// NeuroPLC — Auto-generated IEC 61131-3 SCL
// Graph: mlp | Target: S71200Backend
// Work memory: 75KB | LUT points: 15
// Nodes: 8 | Ops: {'matmul': 4, 'standard_act': 2, 'softmax': 1, 'argmax': 1}


DATA_BLOCK "NeuroPLC_Weights"
{ S7_Optimized_Access := 'TRUE' }
VERSION : 0.1
NON_RETAIN

   // MatMul 'fc0': W(32×28) + b(32)
   w0 : Array[0..927] of Real :=
    -0.1798824, -0.3872150, 0.2042089, 0.0008930, 0.2428655, -0.4397896, 0.1184483, 0.1381282,
    0.0788599, -0.0335890, 0.3613543, -0.3164068, -0.3411417, -0.1364205, -0.3815753, 0.0980671,
    0.0654392, -0.0128052, 0.1792001, -0.1123531, -0.3475231, 0.1503572, -0.0112453, 0.1635510,
    0.1945115, 0.0545633, 0.4145930, -0.3514731, 0.0562777, 0.1928302, -0.1798587, -0.2800348,
    0.1141335, 0.3939485, -0.1134134, -0.3142068, 0.0689715, 0.2764131, -0.3031770, 0.3679943,
    0.0101338, -0.2268585, -0.1187166, 0.4428278, 0.1090220, -0.1324965, -0.4557532, 0.0609620,
    0.2945257, -0.4372934, -0.2674722, 0.2719050, -0.1746262, -0.4510055, -0.2193495, -0.0693161,
    -0.4133973, 0.4597808, 0.3899092, 0.2787638, 0.2211191, -0.2335375, -0.1846817, -0.1514431,
    0.2064924, -0.2602171, 0.2605978, 0.0973142, -0.3398410, -0.4581998, -0.2922807, -0.4378471,
    0.1851701, 0.3957313, 0.2401366, -0.3643467, -0.3337855, 0.0937589, -0.4046761, 0.3407934,
    -0.0060355, 0.0787147, -0.1516189, 0.4190823, 0.1787451, 0.3653978, -0.2563615, -0.3936344,
    -0.4418108, 0.0399490, -0.0161863, 0.3734512, -0.1328384, -0.3586327, 0.0832884, 0.3898760,
    0.0422331, 0.3219765, 0.4136791, 0.4541050, -0.2442907, 0.1221973, -0.3816552, -0.4393946,
    0.4381784, -0.3776088, -0.0355673, 0.0102973, 0.2750401, 0.4402033, -0.0992043, 0.3619939,
    -0.3341672, 0.3641900, 0.0646533, -0.0329038, -0.0519513, 0.4624202, 0.3974202, -0.4135628,
    -0.1883360, 0.1582608, -0.3120753, 0.3418854, -0.1363405, 0.3182234, 0.3987226, -0.2059435,
    0.1484261, 0.1623119, -0.1709910, 0.4116440, 0.4557955, 0.0284270, -0.0647671, 0.4628531,
    -0.4262170, -0.0586162, -0.0261355, 0.3885587, -0.0612076, 0.3511490, -0.4214011, 0.2382351,
    -0.0945188, 0.3279837, -0.4308659, 0.2451999, -0.3082491, -0.0678181, -0.2555402, 0.4352351,
    0.3423308, 0.1892392, -0.4397568, 0.0099074, 0.2687223, -0.4212352, -0.0019993, 0.0687157,
    0.0788325, 0.4018357, 0.4349293, -0.3687074, 0.2395242, 0.3815289, -0.4383415, -0.0245892,
    0.2103941, 0.0996155, 0.1315596, 0.1972513, 0.0423024, 0.3604410, 0.2333128, 0.2266048,
    0.0023598, 0.4544540, -0.2608073, -0.0723180, 0.3625811, 0.1550818, -0.0214169, 0.2343462,
    -0.1961621, -0.1105413, 0.2337353, -0.1424153, 0.1907276, 0.3494135, -0.0083467, 0.4288842,
    -0.3255468, 0.3000529, 0.0926455, -0.1673206, -0.3672895, 0.1358729, 0.2354838, 0.1842398,
    -0.4585243, 0.1047035, 0.4363481, -0.0628617, 0.2278247, -0.2126990, 0.3717730, -0.0640112,
    0.0724800, -0.0195458, -0.3975703, 0.1723518, -0.1848394, 0.1246089, 0.1176429, 0.2367536,
    0.3811733, -0.0844081, 0.0848516, 0.1357539, 0.1603549, -0.0649198, 0.2428739, -0.0198655,
    0.4053905, -0.1223456, -0.0659270, 0.0178697, -0.4600478, -0.0371867, 0.2131490, -0.2711017,
    0.0274099, -0.4619421, 0.1915725, -0.3647681, 0.3060995, -0.1828033, -0.0930496, -0.1906816,
    0.3667245, 0.2526176, 0.2564827, -0.4150518, -0.0207649, 0.2484731, 0.1660505, -0.4234236,
    0.2408383, 0.3804899, 0.3447544, 0.1707152, 0.1783941, -0.0014429, -0.1875186, -0.2965577,
    0.1534259, -0.2261023, 0.2194902, -0.2951540, 0.1165963, 0.2512621, -0.1238675, -0.3037129,
    0.0659142, -0.1324515, 0.4614896, -0.0567672, 0.2121246, -0.2022142, -0.1916900, -0.1399919,
    0.2014992, 0.2298595, -0.3341886, 0.0706455, -0.1369110, -0.3168303, 0.0429791, -0.2362251,
    -0.0745739, 0.1798494, 0.0477831, 0.0812451, -0.0316164, 0.2238211, 0.2806063, 0.4107116,
    -0.2567340, -0.4276187, 0.3658891, -0.0029965, 0.2385021, 0.2209736, -0.3392044, 0.0367437,
    -0.1158386, 0.1748889, -0.0366081, 0.4007239, 0.4308980, -0.0382619, -0.0588789, -0.4497080,
    -0.3535805, -0.0557995, 0.0955771, -0.2503242, -0.2239256, -0.3536082, -0.2803831, -0.3018914,
    -0.1723712, -0.2274993, -0.3283549, 0.4021363, 0.2461150, 0.4450812, -0.2053048, -0.2055161,
    -0.2318867, -0.1703070, 0.0964094, 0.0809516, -0.2962120, 0.2930843, -0.3082349, -0.3325216,
    -0.4066818, 0.1775693, 0.1857542, -0.3768227, -0.3596065, 0.2258550, -0.0153895, -0.1320860,
    -0.2996367, 0.2559390, -0.3494278, 0.0460966, 0.2605145, 0.2958114, 0.4310147, 0.0925957,
    -0.3514842, 0.3076686, -0.1279677, 0.3791227, 0.3633242, 0.0838041, -0.4362233, -0.3780071,
    -0.1231436, -0.4463834, 0.0164300, 0.3187222, 0.3441312, -0.2542373, -0.0990560, -0.3081105,
    -0.2630834, 0.2260506, 0.1768997, -0.0270177, 0.3480961, 0.0443915, -0.2549182, -0.3486338,
    0.0508762, 0.4422698, -0.2197354, 0.2342024, -0.1350438, 0.3885897, 0.1344987, -0.1393131,
    -0.3814989, -0.3116193, 0.2165990, -0.0891674, 0.2220011, -0.3017246, -0.2758035, -0.2295784,
    -0.0438049, 0.2353694, 0.1006879, 0.3114667, -0.4139695, 0.2803482, -0.2584317, 0.2274218,
    -0.4590775, 0.0341408, 0.1420062, -0.3612165, 0.2551019, -0.3598566, 0.0168635, 0.1333762,
    -0.3440666, -0.1630675, -0.0074021, 0.1552494, -0.3977006, -0.1158084, -0.4566253, -0.2927574,
    0.2994344, -0.1632405, -0.3713973, 0.1991937, 0.3783970, -0.2852390, -0.2191832, 0.1243669,
    -0.2800826, 0.3987867, 0.1284276, -0.2516311, -0.3074383, -0.2054294, 0.4527646, -0.1350761,
    -0.3042216, 0.2219902, -0.3400428, -0.2147399, -0.4120946, -0.2263213, -0.0402286, 0.0675365,
    -0.0935789, -0.2593489, 0.0446626, -0.3721133, 0.1265022, 0.4189466, -0.1728224, -0.1179273,
    0.3805940, -0.3371864, -0.3536517, -0.2936776, 0.1048452, 0.1751010, 0.0314007, -0.2069055,
    0.4502559, 0.2475657, -0.0082295, 0.2770777, -0.2011564, -0.4476818, 0.2250594, -0.0451194,
    0.0481762, 0.0532525, 0.3160789, -0.0272306, 0.3712846, 0.4302236, 0.3572811, 0.4566004,
    0.2623333, 0.1703486, -0.0654685, 0.1294028, -0.0769639, -0.0270760, 0.2630037, -0.2648183,
    0.4194202, -0.1575344, -0.3040413, -0.1966138, 0.4314119, 0.1464170, -0.1021344, -0.3179685,
    0.1126420, -0.0385810, -0.3806081, -0.0698207, -0.1330167, -0.4490275, -0.4418296, 0.2836757,
    -0.1377274, -0.0933325, 0.4329276, -0.4006235, 0.2522748, -0.4200759, -0.1706768, -0.3299450,
    -0.4315466, -0.3424816, -0.2155624, -0.3585908, 0.0626948, 0.3521276, -0.3399193, 0.1140631,
    0.0353486, -0.3164425, 0.2124901, 0.3166362, 0.2992722, -0.3527309, -0.4400650, 0.3753791,
    0.3243480, 0.1887977, -0.0438223, 0.4376999, 0.0172825, -0.3287519, -0.4412819, -0.3646971,
    0.3308842, 0.3182985, -0.4211053, -0.3652248, 0.1769410, 0.3722700, -0.3471490, 0.3193542,
    0.2106637, -0.3337017, 0.1720030, -0.2288405, 0.3493201, 0.3209686, 0.2567327, -0.0732017,
    0.2477416, -0.2519081, 0.4488983, 0.1495019, -0.0977263, -0.0334900, 0.0659838, -0.3345148,
    -0.2443900, 0.4558750, 0.2999907, 0.3007113, 0.3972855, 0.2753888, -0.0053852, 0.2395945,
    0.0091295, 0.1445611, -0.2055198, 0.3476967, 0.0850739, 0.3044655, -0.3069745, -0.0617332,
    -0.0156422, 0.1776300, -0.1287701, 0.4349906, 0.1167390, 0.2100853, 0.0931867, 0.2746978,
    -0.0138514, 0.0046518, -0.3086003, -0.1888119, -0.2149056, 0.1065192, 0.2063123, 0.0602527,
    0.2010927, -0.4011554, 0.4382411, -0.0098462, 0.0649581, -0.4081854, -0.3965929, 0.2880442,
    -0.2432063, 0.1212588, -0.3484353, 0.3162225, -0.2948503, -0.4034396, 0.0343257, 0.4352673,
    -0.2021646, -0.3268804, 0.3754787, -0.3476407, -0.4512426, -0.3891115, -0.0950877, 0.0014113,
    -0.3801025, -0.2888759, 0.2253144, 0.2486498, 0.2485408, 0.1874636, -0.1148008, -0.1764733,
    -0.1985060, -0.3856240, -0.1309699, -0.3369353, -0.0277346, -0.3729976, -0.0744570, 0.3116948,
    -0.4212885, -0.2217838, 0.0168743, 0.0647131, -0.2672148, 0.3236766, -0.0746557, -0.4231054,
    0.1975563, 0.1557159, 0.0349012, -0.3396184, -0.1297497, -0.4186305, -0.0316620, -0.0924572,
    -0.4292775, 0.3364194, 0.2239106, 0.4233520, -0.2597517, 0.1058979, 0.0360005, -0.0301330,
    -0.2367468, -0.3565944, 0.4520262, -0.0556437, -0.0790337, 0.1684058, 0.0914626, -0.0453906,
    0.3796009, -0.2842137, -0.3293831, -0.1658794, -0.4397863, 0.2365771, 0.0294120, 0.4533179,
    -0.0859124, -0.0621766, 0.3045017, -0.3232293, 0.2738206, -0.0116338, 0.3944798, -0.2239275,
    0.2238147, -0.2989884, 0.3236126, -0.4262000, -0.3253698, 0.1608732, 0.3702686, 0.1019678,
    -0.2107479, -0.2611701, 0.4136789, 0.0865699, 0.4570325, 0.2902318, -0.1133356, 0.2509187,
    -0.3027558, -0.0267411, 0.4365703, 0.4290322, 0.0391642, -0.1402205, -0.2419274, 0.3942315,
    -0.3281853, 0.3526350, -0.2294700, -0.0201786, -0.4453179, 0.0182093, 0.0901008, 0.0272455,
    0.0261993, -0.0577734, -0.1454998, -0.1999438, 0.3330531, 0.1162911, -0.1408730, 0.3945518,
    0.0200893, 0.3864298, 0.3662851, -0.4315742, 0.4240045, 0.0685083, -0.0862473, 0.1716394,
    -0.0252949, -0.1983226, -0.0851686, 0.0366299, 0.3082128, 0.3418522, 0.0999441, -0.3636666,
    -0.0260158, 0.4472989, -0.1166421, 0.0326859, -0.0569831, 0.2964681, 0.3741921, 0.0694074,
    -0.2019286, -0.2991379, 0.1687691, -0.1963241, -0.2953035, -0.4300376, -0.2427881, 0.0319568,
    -0.2237948, 0.3365344, -0.2773279, 0.1702439, -0.2662200, -0.4590583, 0.1108428, 0.2470049,
    -0.3626023, 0.1612943, 0.0753302, -0.1507791, 0.3780867, 0.2598709, 0.2767858, -0.1879475,
    -0.1899060, -0.4502818, -0.3476299, 0.2807263, 0.2010535, -0.2459695, 0.0484484, 0.2529786,
    -0.4405471, -0.0633909, 0.3059275, 0.1004434, 0.0873103, 0.1176765, -0.0138679, 0.3308610,
    -0.1480782, 0.3191504, 0.3431600, 0.0682138, -0.3328019, 0.1721126, 0.1514601, 0.1276880,
    0.3282012, 0.1886778, -0.2926646, -0.3705381, 0.3847846, 0.1586861, -0.2964849, -0.2298914,
    0.3726317, -0.2340294, -0.3934847, 0.3866403, 0.3287364, -0.4364095, 0.3202796, -0.4572898,
    0.4240396, 0.2946174, 0.4263544, -0.3875704, -0.2983319, 0.2481298, -0.3679308, 0.3585340,
    -0.2879644, 0.1617320, 0.2525170, 0.4445124, -0.3569905, 0.3035758, 0.3973208, -0.3388606,
    0.1971553, 0.4202124, -0.0093552, -0.2728116, 0.4091376, 0.3026397, -0.1690369, -0.1815633,
    -0.3018734, 0.1926507, -0.1460906, -0.4044804, 0.3854034, 0.2598969, 0.0819964, 0.0040537,
    0.0088892, 0.1276613, -0.0934737, -0.0725756, 0.3761741, 0.1721867, -0.0835514, -0.3227195,
    -0.1970350, -0.1828245, -0.2169749, 0.1113454, 0.2208307, -0.2727543, -0.2885212, 0.4582173,
    0.1132768, 0.0894297, -0.1760622, -0.4032561, -0.1639080, -0.4546085, -0.1885196, 0.2742654,
    0.3573460, -0.0079773, 0.3492272, 0.0432554, -0.0694141, -0.0292612, 0.0648459, 0.0404633,
    0.0550900, -0.0040946, -0.0961987, 0.3513191, -0.3384297, -0.3327979, -0.2216373, -0.1413240,
    -0.0152824, -0.4382769, 0.3047727, -0.3338848, -0.0337600, -0.2625723, -0.3748975, -0.1234908,
    0.2812771, -0.0338805, 0.0630252, 0.2799799, -0.1394900, 0.3232564, -0.2665378, 0.2301099,
    -0.1728424, 0.3568045, 0.1587069, -0.1994252, 0.1759624, -0.2301375, 0.0293344, 0.2550743,
    0.1888990, 0.2785141, 0.2414417, 0.1385446, 0.2032104, -0.3619106, -0.1416969, 0.3761026,
    0.0, 0.0, 0.0, 0.0, 0.0, 0.0, 0.0, 0.0,
    0.0, 0.0, 0.0, 0.0, 0.0, 0.0, 0.0, 0.0,
    0.0, 0.0, 0.0, 0.0, 0.0, 0.0, 0.0, 0.0,
    0.0, 0.0, 0.0, 0.0, 0.0, 0.0, 0.0, 0.0;

   // MatMul 'fc1': W(16×32) + b(16)
   w1 : Array[0..527] of Real :=
    -0.1841003, -0.3950176, 0.0280379, 0.0440260, 0.1147591, 0.2946690, -0.1696201, 0.0702065,
    -0.1734065, -0.0780731, 0.1729136, -0.2214055, 0.1615332, -0.1130018, 0.1126955, -0.1627842,
    -0.2089999, 0.0900196, -0.2156965, -0.0010487, 0.3421980, -0.3204773, -0.1042151, 0.2794774,
    0.1362123, -0.1695349, -0.3630999, -0.2400454, -0.3631713, -0.2607281, 0.4220854, -0.2033405,
    0.4245700, 0.4134347, 0.2165404, -0.3439045, 0.4052791, -0.0289224, 0.0352862, -0.2532949,
    0.0514103, -0.1915463, -0.1317405, 0.1894104, -0.1309697, 0.4199851, -0.2161604, 0.1424241,
    -0.0695876, 0.0812146, -0.3267484, 0.1127291, 0.0712753, 0.0544753, 0.2083792, 0.4198444,
    -0.0903308, 0.4007897, -0.3954699, -0.0837158, -0.2097752, 0.0160278, -0.4290526, -0.0252581,
    -0.2535323, 0.3457471, 0.2822391, 0.3988800, 0.1782279, 0.0142821, 0.2393648, -0.1553738,
    0.4060715, 0.4100494, -0.3253954, -0.3813735, 0.4294659, 0.2282157, -0.1696985, -0.3954830,
    -0.1343698, 0.0225449, 0.3071480, 0.1503303, 0.2892320, -0.3464375, 0.3547571, -0.3604251,
    -0.2291267, 0.0886436, 0.3920235, -0.3591582, 0.1108168, 0.3186001, 0.3305989, -0.1636246,
    -0.4108425, -0.0282269, 0.2816935, -0.3807812, 0.0377470, 0.1486996, 0.1058756, -0.3785081,
    0.1195602, -0.1099812, -0.2850332, -0.2532795, 0.2460700, 0.1802454, 0.3887673, 0.3546645,
    0.1356663, -0.4002051, 0.1958930, 0.3444175, -0.2449986, -0.0592304, 0.2936576, 0.0734874,
    -0.3506431, 0.0448850, 0.1267957, -0.0889452, -0.1783398, 0.4244988, -0.0005950, -0.2101975,
    0.0582885, 0.0898391, 0.0216084, 0.3572374, -0.3613801, -0.1606691, -0.2318281, 0.2716186,
    -0.0560970, 0.2975237, -0.3013628, -0.1173695, -0.3505674, 0.1472747, 0.0306037, 0.1608355,
    -0.3668388, 0.1993875, -0.1024434, -0.3948376, 0.2310698, 0.0110251, 0.2700239, -0.3990251,
    -0.3589656, 0.3225909, 0.3532399, -0.3362035, 0.2659501, -0.2563055, -0.3352330, 0.3330118,
    -0.3832548, 0.2277593, -0.2611139, 0.1635678, 0.3083868, 0.3321955, -0.0756106, -0.4202253,
    -0.4210085, 0.0254245, 0.4143491, 0.0979612, 0.0923779, 0.0762489, -0.1803973, -0.1762412,
    -0.1601437, 0.2343485, -0.2330645, -0.4151017, -0.4032581, -0.2181285, -0.1266952, 0.2701829,
    0.3503337, 0.3371424, 0.0500940, -0.0518085, -0.3143240, -0.2576985, 0.0838322, -0.0579774,
    -0.2055396, 0.4009449, 0.0156569, -0.2904895, -0.2681209, -0.0107362, 0.0463802, -0.2953869,
    0.4148783, -0.3537356, -0.0661243, 0.2925996, 0.0898428, 0.4177988, 0.3496406, -0.3616090,
    0.2731358, 0.0594644, -0.2220350, 0.3457292, -0.0209776, 0.0297440, 0.2737146, 0.3270914,
    -0.3035161, 0.0231363, -0.2473483, 0.3730231, 0.2400877, 0.1128676, 0.0010069, -0.2103814,
    -0.0423518, 0.1287846, -0.2755486, 0.2502011, -0.3502574, 0.0082882, 0.2342134, -0.2862676,
    0.3997168, 0.2841206, 0.3299266, -0.1131397, -0.2668519, -0.2157065, 0.3389430, -0.2941397,
    0.4323460, -0.0482011, 0.1886959, -0.2788211, 0.3894212, 0.1545921, 0.3432020, -0.1336565,
    0.2985416, 0.2803046, -0.2245447, -0.2217844, 0.4067388, -0.3139164, 0.3276515, 0.3778521,
    0.0466528, 0.0636986, -0.3395925, 0.3690981, -0.2149493, -0.2441782, -0.3498707, 0.0939149,
    -0.3066922, -0.1904545, -0.4194795, 0.0577288, -0.0715801, 0.2936807, 0.3827896, -0.1505448,
    -0.2847440, -0.1595511, 0.0994487, 0.0144897, -0.3030011, -0.0394793, -0.3570347, -0.0396204,
    0.1410332, -0.3515431, -0.2199971, 0.2524821, 0.1527711, 0.2854764, -0.0980022, -0.3928814,
    0.4188430, -0.2180078, -0.3378795, -0.2400968, 0.0973825, -0.4067127, -0.3336179, -0.1964155,
    0.3282059, -0.1130220, -0.4168500, 0.4280160, 0.1311055, -0.3648337, -0.4253438, 0.2005218,
    -0.1747648, 0.0874954, -0.1753466, 0.1078633, 0.0307744, 0.2767422, 0.2746042, 0.1012669,
    -0.4009462, 0.3802539, -0.4298933, 0.2958619, -0.3853600, -0.0928518, 0.0112549, -0.2410028,
    -0.1998202, -0.1247788, -0.2532034, -0.1840077, -0.0097570, 0.0498497, 0.1501264, -0.1523731,
    0.1660306, 0.3964193, 0.0149433, 0.2128017, -0.1015208, 0.2488470, -0.3308116, 0.1322182,
    0.0452061, -0.2983263, 0.2222392, -0.0971295, -0.1187560, -0.2245519, 0.2802809, 0.4223242,
    0.2730812, -0.0907452, 0.2778142, 0.0116081, 0.2301807, 0.0370663, -0.1044484, -0.1732805,
    0.2800431, -0.1159531, -0.1670154, -0.0533327, 0.1396156, 0.3444407, -0.0747188, -0.3951142,
    -0.0871275, 0.3335563, -0.0700926, -0.0987261, -0.0334665, -0.1378284, -0.1616814, 0.3731155,
    -0.3847730, -0.2036186, 0.4113233, -0.2007953, 0.1136580, 0.0199758, -0.1730417, -0.2137244,
    0.3787228, 0.2845047, -0.0253214, 0.0397584, -0.1338087, 0.3907075, 0.0293069, -0.1894936,
    0.2623669, -0.1419247, 0.1988509, 0.3641036, 0.4179319, 0.0193644, -0.3016763, -0.2553127,
    0.0341927, -0.2933192, 0.3224567, -0.0938100, -0.4136013, -0.0439183, 0.1660686, 0.3230760,
    -0.2442258, -0.4120509, -0.2696367, -0.2744891, 0.0259897, -0.2600366, 0.1869681, 0.2555002,
    -0.1946192, -0.1122633, -0.4029176, -0.0710380, 0.3222395, -0.2946250, 0.2944258, 0.1149372,
    0.1621488, -0.3521335, -0.1484178, -0.2395614, 0.2510083, -0.0162863, 0.3919969, -0.4237986,
    0.1645654, -0.1310851, 0.2434124, 0.2159853, -0.0879131, -0.0384991, 0.2112199, 0.1240114,
    -0.2128599, -0.1464353, 0.2506914, 0.3504371, 0.0575993, -0.1435232, -0.0928054, -0.3425918,
    -0.1951562, 0.0662211, -0.0652936, 0.3474210, 0.3170411, 0.3430875, 0.0670799, -0.1089404,
    -0.3778215, -0.2251768, 0.4261730, -0.3357262, -0.1937545, 0.2503859, 0.1622876, -0.3160965,
    0.1899634, -0.3406923, -0.0890604, 0.1557132, 0.0973966, -0.4325262, -0.1982196, -0.1852470,
    -0.0401643, 0.2625172, 0.1903876, -0.4238683, 0.1880887, 0.1010092, -0.3720742, -0.0422780,
    0.2044589, 0.2732541, -0.2875984, -0.1535293, -0.0050445, 0.1866603, -0.1373991, -0.3727299,
    -0.1867637, -0.4104604, -0.1678579, -0.1667786, -0.1890316, -0.3301499, -0.1857497, 0.2939049,
    -0.0040281, 0.1575826, 0.1627137, 0.2202530, -0.0844541, -0.0894054, -0.3965610, 0.0585302,
    -0.0476493, 0.1316660, -0.2428709, -0.0171687, -0.1816288, 0.4306199, -0.0929443, -0.1739965,
    -0.1473018, -0.1209739, 0.3987128, -0.3711412, 0.1341918, -0.2781068, -0.0634658, -0.2352583,
    0.0, 0.0, 0.0, 0.0, 0.0, 0.0, 0.0, 0.0,
    0.0, 0.0, 0.0, 0.0, 0.0, 0.0, 0.0, 0.0;

   // MatMul 'fc2': W(4×16) + b(4)
   w2 : Array[0..67] of Real :=
    0.1326775, -0.5272908, 0.0543207, -0.0181786, 0.2338884, 0.4969643, 0.2776969, 0.2249198,
    0.1608169, -0.4576403, 0.5489935, 0.1290960, 0.0282424, -0.4624947, -0.4523918, -0.5721835,
    -0.4659075, -0.0712391, -0.4551743, -0.3424331, -0.1415611, -0.5302606, -0.2768892, 0.2787506,
    0.2798988, 0.2107574, 0.4792312, 0.4036999, -0.0253411, -0.5930076, 0.4648258, -0.3432639,
    0.1270192, 0.2098873, -0.1395269, 0.1806177, -0.3960660, -0.4025090, 0.1715716, 0.2829821,
    -0.0803854, -0.5585088, -0.6079782, -0.4716686, 0.5347964, -0.5765373, -0.1166642, -0.2985954,
    -0.3982801, -0.1811747, 0.0273219, 0.1674641, 0.1254434, 0.4325371, 0.3858762, 0.4819646,
    -0.3050049, 0.1955859, 0.2508789, -0.3311853, 0.5485005, 0.2929417, 0.3204345, -0.3687590,
    0.0, 0.0, 0.0, 0.0;

   // Total: 3 array blocks
END_DATA_BLOCK

FUNCTION_BLOCK "NeuroPLC_Inference"
{ S7_Optimized_Access := 'TRUE' }
VERSION : 0.1
VAR_INPUT
    features : Array[0..27] of Real;
END_VAR

VAR_OUTPUT
    fault_class : Int;
    confidence : Real;
END_VAR

VAR
    i, j, k : Int;
    sum_val, max_val, t_val : Real;
    v0 : Array[0..27] of Real;
    v1 : Array[0..31] of Real;
    v2 : Array[0..31] of Real;
    v3 : Array[0..15] of Real;
    v4 : Array[0..15] of Real;
    v5 : Array[0..3] of Real;
    v6 : Array[0..3] of Real;
END_VAR

BEGIN
    // ---- Input ----
    FOR i := 0 TO 27 DO
        v0[i] := features[i];
    END_FOR;

    // ---- fc0: MatMul(28→32) ----
    // W = "NeuroPLC_Weights".w0[:896],   b = w0[896:]
    v1[0] := "NeuroPLC_Weights".w0[896 + 0] + "NeuroPLC_Weights".w0[0] * v0[0] + "NeuroPLC_Weights".w0[1] * v0[1] + "NeuroPLC_Weights".w0[2] * v0[2] + "NeuroPLC_Weights".w0[3] * v0[3] + "NeuroPLC_Weights".w0[4] * v0[4] + "NeuroPLC_Weights".w0[5] * v0[5] + "NeuroPLC_Weights".w0[6] * v0[6] + "NeuroPLC_Weights".w0[7] * v0[7] + "NeuroPLC_Weights".w0[8] * v0[8] + "NeuroPLC_Weights".w0[9] * v0[9] + "NeuroPLC_Weights".w0[10] * v0[10] + "NeuroPLC_Weights".w0[11] * v0[11] + "NeuroPLC_Weights".w0[12] * v0[12] + "NeuroPLC_Weights".w0[13] * v0[13] + "NeuroPLC_Weights".w0[14] * v0[14] + "NeuroPLC_Weights".w0[15] * v0[15] + "NeuroPLC_Weights".w0[16] * v0[16] + "NeuroPLC_Weights".w0[17] * v0[17] + "NeuroPLC_Weights".w0[18] * v0[18] + "NeuroPLC_Weights".w0[19] * v0[19] + "NeuroPLC_Weights".w0[20] * v0[20] + "NeuroPLC_Weights".w0[21] * v0[21] + "NeuroPLC_Weights".w0[22] * v0[22] + "NeuroPLC_Weights".w0[23] * v0[23] + "NeuroPLC_Weights".w0[24] * v0[24] + "NeuroPLC_Weights".w0[25] * v0[25] + "NeuroPLC_Weights".w0[26] * v0[26] + "NeuroPLC_Weights".w0[27] * v0[27];
    v1[1] := "NeuroPLC_Weights".w0[896 + 1] + "NeuroPLC_Weights".w0[28] * v0[0] + "NeuroPLC_Weights".w0[29] * v0[1] + "NeuroPLC_Weights".w0[30] * v0[2] + "NeuroPLC_Weights".w0[31] * v0[3] + "NeuroPLC_Weights".w0[32] * v0[4] + "NeuroPLC_Weights".w0[33] * v0[5] + "NeuroPLC_Weights".w0[34] * v0[6] + "NeuroPLC_Weights".w0[35] * v0[7] + "NeuroPLC_Weights".w0[36] * v0[8] + "NeuroPLC_Weights".w0[37] * v0[9] + "NeuroPLC_Weights".w0[38] * v0[10] + "NeuroPLC_Weights".w0[39] * v0[11] + "NeuroPLC_Weights".w0[40] * v0[12] + "NeuroPLC_Weights".w0[41] * v0[13] + "NeuroPLC_Weights".w0[42] * v0[14] + "NeuroPLC_Weights".w0[43] * v0[15] + "NeuroPLC_Weights".w0[44] * v0[16] + "NeuroPLC_Weights".w0[45] * v0[17] + "NeuroPLC_Weights".w0[46] * v0[18] + "NeuroPLC_Weights".w0[47] * v0[19] + "NeuroPLC_Weights".w0[48] * v0[20] + "NeuroPLC_Weights".w0[49] * v0[21] + "NeuroPLC_Weights".w0[50] * v0[22] + "NeuroPLC_Weights".w0[51] * v0[23] + "NeuroPLC_Weights".w0[52] * v0[24] + "NeuroPLC_Weights".w0[53] * v0[25] + "NeuroPLC_Weights".w0[54] * v0[26] + "NeuroPLC_Weights".w0[55] * v0[27];
    v1[2] := "NeuroPLC_Weights".w0[896 + 2] + "NeuroPLC_Weights".w0[56] * v0[0] + "NeuroPLC_Weights".w0[57] * v0[1] + "NeuroPLC_Weights".w0[58] * v0[2] + "NeuroPLC_Weights".w0[59] * v0[3] + "NeuroPLC_Weights".w0[60] * v0[4] + "NeuroPLC_Weights".w0[61] * v0[5] + "NeuroPLC_Weights".w0[62] * v0[6] + "NeuroPLC_Weights".w0[63] * v0[7] + "NeuroPLC_Weights".w0[64] * v0[8] + "NeuroPLC_Weights".w0[65] * v0[9] + "NeuroPLC_Weights".w0[66] * v0[10] + "NeuroPLC_Weights".w0[67] * v0[11] + "NeuroPLC_Weights".w0[68] * v0[12] + "NeuroPLC_Weights".w0[69] * v0[13] + "NeuroPLC_Weights".w0[70] * v0[14] + "NeuroPLC_Weights".w0[71] * v0[15] + "NeuroPLC_Weights".w0[72] * v0[16] + "NeuroPLC_Weights".w0[73] * v0[17] + "NeuroPLC_Weights".w0[74] * v0[18] + "NeuroPLC_Weights".w0[75] * v0[19] + "NeuroPLC_Weights".w0[76] * v0[20] + "NeuroPLC_Weights".w0[77] * v0[21] + "NeuroPLC_Weights".w0[78] * v0[22] + "NeuroPLC_Weights".w0[79] * v0[23] + "NeuroPLC_Weights".w0[80] * v0[24] + "NeuroPLC_Weights".w0[81] * v0[25] + "NeuroPLC_Weights".w0[82] * v0[26] + "NeuroPLC_Weights".w0[83] * v0[27];
    v1[3] := "NeuroPLC_Weights".w0[896 + 3] + "NeuroPLC_Weights".w0[84] * v0[0] + "NeuroPLC_Weights".w0[85] * v0[1] + "NeuroPLC_Weights".w0[86] * v0[2] + "NeuroPLC_Weights".w0[87] * v0[3] + "NeuroPLC_Weights".w0[88] * v0[4] + "NeuroPLC_Weights".w0[89] * v0[5] + "NeuroPLC_Weights".w0[90] * v0[6] + "NeuroPLC_Weights".w0[91] * v0[7] + "NeuroPLC_Weights".w0[92] * v0[8] + "NeuroPLC_Weights".w0[93] * v0[9] + "NeuroPLC_Weights".w0[94] * v0[10] + "NeuroPLC_Weights".w0[95] * v0[11] + "NeuroPLC_Weights".w0[96] * v0[12] + "NeuroPLC_Weights".w0[97] * v0[13] + "NeuroPLC_Weights".w0[98] * v0[14] + "NeuroPLC_Weights".w0[99] * v0[15] + "NeuroPLC_Weights".w0[100] * v0[16] + "NeuroPLC_Weights".w0[101] * v0[17] + "NeuroPLC_Weights".w0[102] * v0[18] + "NeuroPLC_Weights".w0[103] * v0[19] + "NeuroPLC_Weights".w0[104] * v0[20] + "NeuroPLC_Weights".w0[105] * v0[21] + "NeuroPLC_Weights".w0[106] * v0[22] + "NeuroPLC_Weights".w0[107] * v0[23] + "NeuroPLC_Weights".w0[108] * v0[24] + "NeuroPLC_Weights".w0[109] * v0[25] + "NeuroPLC_Weights".w0[110] * v0[26] + "NeuroPLC_Weights".w0[111] * v0[27];
    v1[4] := "NeuroPLC_Weights".w0[896 + 4] + "NeuroPLC_Weights".w0[112] * v0[0] + "NeuroPLC_Weights".w0[113] * v0[1] + "NeuroPLC_Weights".w0[114] * v0[2] + "NeuroPLC_Weights".w0[115] * v0[3] + "NeuroPLC_Weights".w0[116] * v0[4] + "NeuroPLC_Weights".w0[117] * v0[5] + "NeuroPLC_Weights".w0[118] * v0[6] + "NeuroPLC_Weights".w0[119] * v0[7] + "NeuroPLC_Weights".w0[120] * v0[8] + "NeuroPLC_Weights".w0[121] * v0[9] + "NeuroPLC_Weights".w0[122] * v0[10] + "NeuroPLC_Weights".w0[123] * v0[11] + "NeuroPLC_Weights".w0[124] * v0[12] + "NeuroPLC_Weights".w0[125] * v0[13] + "NeuroPLC_Weights".w0[126] * v0[14] + "NeuroPLC_Weights".w0[127] * v0[15] + "NeuroPLC_Weights".w0[128] * v0[16] + "NeuroPLC_Weights".w0[129] * v0[17] + "NeuroPLC_Weights".w0[130] * v0[18] + "NeuroPLC_Weights".w0[131] * v0[19] + "NeuroPLC_Weights".w0[132] * v0[20] + "NeuroPLC_Weights".w0[133] * v0[21] + "NeuroPLC_Weights".w0[134] * v0[22] + "NeuroPLC_Weights".w0[135] * v0[23] + "NeuroPLC_Weights".w0[136] * v0[24] + "NeuroPLC_Weights".w0[137] * v0[25] + "NeuroPLC_Weights".w0[138] * v0[26] + "NeuroPLC_Weights".w0[139] * v0[27];
    v1[5] := "NeuroPLC_Weights".w0[896 + 5] + "NeuroPLC_Weights".w0[140] * v0[0] + "NeuroPLC_Weights".w0[141] * v0[1] + "NeuroPLC_Weights".w0[142] * v0[2] + "NeuroPLC_Weights".w0[143] * v0[3] + "NeuroPLC_Weights".w0[144] * v0[4] + "NeuroPLC_Weights".w0[145] * v0[5] + "NeuroPLC_Weights".w0[146] * v0[6] + "NeuroPLC_Weights".w0[147] * v0[7] + "NeuroPLC_Weights".w0[148] * v0[8] + "NeuroPLC_Weights".w0[149] * v0[9] + "NeuroPLC_Weights".w0[150] * v0[10] + "NeuroPLC_Weights".w0[151] * v0[11] + "NeuroPLC_Weights".w0[152] * v0[12] + "NeuroPLC_Weights".w0[153] * v0[13] + "NeuroPLC_Weights".w0[154] * v0[14] + "NeuroPLC_Weights".w0[155] * v0[15] + "NeuroPLC_Weights".w0[156] * v0[16] + "NeuroPLC_Weights".w0[157] * v0[17] + "NeuroPLC_Weights".w0[158] * v0[18] + "NeuroPLC_Weights".w0[159] * v0[19] + "NeuroPLC_Weights".w0[160] * v0[20] + "NeuroPLC_Weights".w0[161] * v0[21] + "NeuroPLC_Weights".w0[162] * v0[22] + "NeuroPLC_Weights".w0[163] * v0[23] + "NeuroPLC_Weights".w0[164] * v0[24] + "NeuroPLC_Weights".w0[165] * v0[25] + "NeuroPLC_Weights".w0[166] * v0[26] + "NeuroPLC_Weights".w0[167] * v0[27];
    v1[6] := "NeuroPLC_Weights".w0[896 + 6] + "NeuroPLC_Weights".w0[168] * v0[0] + "NeuroPLC_Weights".w0[169] * v0[1] + "NeuroPLC_Weights".w0[170] * v0[2] + "NeuroPLC_Weights".w0[171] * v0[3] + "NeuroPLC_Weights".w0[172] * v0[4] + "NeuroPLC_Weights".w0[173] * v0[5] + "NeuroPLC_Weights".w0[174] * v0[6] + "NeuroPLC_Weights".w0[175] * v0[7] + "NeuroPLC_Weights".w0[176] * v0[8] + "NeuroPLC_Weights".w0[177] * v0[9] + "NeuroPLC_Weights".w0[178] * v0[10] + "NeuroPLC_Weights".w0[179] * v0[11] + "NeuroPLC_Weights".w0[180] * v0[12] + "NeuroPLC_Weights".w0[181] * v0[13] + "NeuroPLC_Weights".w0[182] * v0[14] + "NeuroPLC_Weights".w0[183] * v0[15] + "NeuroPLC_Weights".w0[184] * v0[16] + "NeuroPLC_Weights".w0[185] * v0[17] + "NeuroPLC_Weights".w0[186] * v0[18] + "NeuroPLC_Weights".w0[187] * v0[19] + "NeuroPLC_Weights".w0[188] * v0[20] + "NeuroPLC_Weights".w0[189] * v0[21] + "NeuroPLC_Weights".w0[190] * v0[22] + "NeuroPLC_Weights".w0[191] * v0[23] + "NeuroPLC_Weights".w0[192] * v0[24] + "NeuroPLC_Weights".w0[193] * v0[25] + "NeuroPLC_Weights".w0[194] * v0[26] + "NeuroPLC_Weights".w0[195] * v0[27];
    v1[7] := "NeuroPLC_Weights".w0[896 + 7] + "NeuroPLC_Weights".w0[196] * v0[0] + "NeuroPLC_Weights".w0[197] * v0[1] + "NeuroPLC_Weights".w0[198] * v0[2] + "NeuroPLC_Weights".w0[199] * v0[3] + "NeuroPLC_Weights".w0[200] * v0[4] + "NeuroPLC_Weights".w0[201] * v0[5] + "NeuroPLC_Weights".w0[202] * v0[6] + "NeuroPLC_Weights".w0[203] * v0[7] + "NeuroPLC_Weights".w0[204] * v0[8] + "NeuroPLC_Weights".w0[205] * v0[9] + "NeuroPLC_Weights".w0[206] * v0[10] + "NeuroPLC_Weights".w0[207] * v0[11] + "NeuroPLC_Weights".w0[208] * v0[12] + "NeuroPLC_Weights".w0[209] * v0[13] + "NeuroPLC_Weights".w0[210] * v0[14] + "NeuroPLC_Weights".w0[211] * v0[15] + "NeuroPLC_Weights".w0[212] * v0[16] + "NeuroPLC_Weights".w0[213] * v0[17] + "NeuroPLC_Weights".w0[214] * v0[18] + "NeuroPLC_Weights".w0[215] * v0[19] + "NeuroPLC_Weights".w0[216] * v0[20] + "NeuroPLC_Weights".w0[217] * v0[21] + "NeuroPLC_Weights".w0[218] * v0[22] + "NeuroPLC_Weights".w0[219] * v0[23] + "NeuroPLC_Weights".w0[220] * v0[24] + "NeuroPLC_Weights".w0[221] * v0[25] + "NeuroPLC_Weights".w0[222] * v0[26] + "NeuroPLC_Weights".w0[223] * v0[27];
    v1[8] := "NeuroPLC_Weights".w0[896 + 8] + "NeuroPLC_Weights".w0[224] * v0[0] + "NeuroPLC_Weights".w0[225] * v0[1] + "NeuroPLC_Weights".w0[226] * v0[2] + "NeuroPLC_Weights".w0[227] * v0[3] + "NeuroPLC_Weights".w0[228] * v0[4] + "NeuroPLC_Weights".w0[229] * v0[5] + "NeuroPLC_Weights".w0[230] * v0[6] + "NeuroPLC_Weights".w0[231] * v0[7] + "NeuroPLC_Weights".w0[232] * v0[8] + "NeuroPLC_Weights".w0[233] * v0[9] + "NeuroPLC_Weights".w0[234] * v0[10] + "NeuroPLC_Weights".w0[235] * v0[11] + "NeuroPLC_Weights".w0[236] * v0[12] + "NeuroPLC_Weights".w0[237] * v0[13] + "NeuroPLC_Weights".w0[238] * v0[14] + "NeuroPLC_Weights".w0[239] * v0[15] + "NeuroPLC_Weights".w0[240] * v0[16] + "NeuroPLC_Weights".w0[241] * v0[17] + "NeuroPLC_Weights".w0[242] * v0[18] + "NeuroPLC_Weights".w0[243] * v0[19] + "NeuroPLC_Weights".w0[244] * v0[20] + "NeuroPLC_Weights".w0[245] * v0[21] + "NeuroPLC_Weights".w0[246] * v0[22] + "NeuroPLC_Weights".w0[247] * v0[23] + "NeuroPLC_Weights".w0[248] * v0[24] + "NeuroPLC_Weights".w0[249] * v0[25] + "NeuroPLC_Weights".w0[250] * v0[26] + "NeuroPLC_Weights".w0[251] * v0[27];
    v1[9] := "NeuroPLC_Weights".w0[896 + 9] + "NeuroPLC_Weights".w0[252] * v0[0] + "NeuroPLC_Weights".w0[253] * v0[1] + "NeuroPLC_Weights".w0[254] * v0[2] + "NeuroPLC_Weights".w0[255] * v0[3] + "NeuroPLC_Weights".w0[256] * v0[4] + "NeuroPLC_Weights".w0[257] * v0[5] + "NeuroPLC_Weights".w0[258] * v0[6] + "NeuroPLC_Weights".w0[259] * v0[7] + "NeuroPLC_Weights".w0[260] * v0[8] + "NeuroPLC_Weights".w0[261] * v0[9] + "NeuroPLC_Weights".w0[262] * v0[10] + "NeuroPLC_Weights".w0[263] * v0[11] + "NeuroPLC_Weights".w0[264] * v0[12] + "NeuroPLC_Weights".w0[265] * v0[13] + "NeuroPLC_Weights".w0[266] * v0[14] + "NeuroPLC_Weights".w0[267] * v0[15] + "NeuroPLC_Weights".w0[268] * v0[16] + "NeuroPLC_Weights".w0[269] * v0[17] + "NeuroPLC_Weights".w0[270] * v0[18] + "NeuroPLC_Weights".w0[271] * v0[19] + "NeuroPLC_Weights".w0[272] * v0[20] + "NeuroPLC_Weights".w0[273] * v0[21] + "NeuroPLC_Weights".w0[274] * v0[22] + "NeuroPLC_Weights".w0[275] * v0[23] + "NeuroPLC_Weights".w0[276] * v0[24] + "NeuroPLC_Weights".w0[277] * v0[25] + "NeuroPLC_Weights".w0[278] * v0[26] + "NeuroPLC_Weights".w0[279] * v0[27];
    v1[10] := "NeuroPLC_Weights".w0[896 + 10] + "NeuroPLC_Weights".w0[280] * v0[0] + "NeuroPLC_Weights".w0[281] * v0[1] + "NeuroPLC_Weights".w0[282] * v0[2] + "NeuroPLC_Weights".w0[283] * v0[3] + "NeuroPLC_Weights".w0[284] * v0[4] + "NeuroPLC_Weights".w0[285] * v0[5] + "NeuroPLC_Weights".w0[286] * v0[6] + "NeuroPLC_Weights".w0[287] * v0[7] + "NeuroPLC_Weights".w0[288] * v0[8] + "NeuroPLC_Weights".w0[289] * v0[9] + "NeuroPLC_Weights".w0[290] * v0[10] + "NeuroPLC_Weights".w0[291] * v0[11] + "NeuroPLC_Weights".w0[292] * v0[12] + "NeuroPLC_Weights".w0[293] * v0[13] + "NeuroPLC_Weights".w0[294] * v0[14] + "NeuroPLC_Weights".w0[295] * v0[15] + "NeuroPLC_Weights".w0[296] * v0[16] + "NeuroPLC_Weights".w0[297] * v0[17] + "NeuroPLC_Weights".w0[298] * v0[18] + "NeuroPLC_Weights".w0[299] * v0[19] + "NeuroPLC_Weights".w0[300] * v0[20] + "NeuroPLC_Weights".w0[301] * v0[21] + "NeuroPLC_Weights".w0[302] * v0[22] + "NeuroPLC_Weights".w0[303] * v0[23] + "NeuroPLC_Weights".w0[304] * v0[24] + "NeuroPLC_Weights".w0[305] * v0[25] + "NeuroPLC_Weights".w0[306] * v0[26] + "NeuroPLC_Weights".w0[307] * v0[27];
    v1[11] := "NeuroPLC_Weights".w0[896 + 11] + "NeuroPLC_Weights".w0[308] * v0[0] + "NeuroPLC_Weights".w0[309] * v0[1] + "NeuroPLC_Weights".w0[310] * v0[2] + "NeuroPLC_Weights".w0[311] * v0[3] + "NeuroPLC_Weights".w0[312] * v0[4] + "NeuroPLC_Weights".w0[313] * v0[5] + "NeuroPLC_Weights".w0[314] * v0[6] + "NeuroPLC_Weights".w0[315] * v0[7] + "NeuroPLC_Weights".w0[316] * v0[8] + "NeuroPLC_Weights".w0[317] * v0[9] + "NeuroPLC_Weights".w0[318] * v0[10] + "NeuroPLC_Weights".w0[319] * v0[11] + "NeuroPLC_Weights".w0[320] * v0[12] + "NeuroPLC_Weights".w0[321] * v0[13] + "NeuroPLC_Weights".w0[322] * v0[14] + "NeuroPLC_Weights".w0[323] * v0[15] + "NeuroPLC_Weights".w0[324] * v0[16] + "NeuroPLC_Weights".w0[325] * v0[17] + "NeuroPLC_Weights".w0[326] * v0[18] + "NeuroPLC_Weights".w0[327] * v0[19] + "NeuroPLC_Weights".w0[328] * v0[20] + "NeuroPLC_Weights".w0[329] * v0[21] + "NeuroPLC_Weights".w0[330] * v0[22] + "NeuroPLC_Weights".w0[331] * v0[23] + "NeuroPLC_Weights".w0[332] * v0[24] + "NeuroPLC_Weights".w0[333] * v0[25] + "NeuroPLC_Weights".w0[334] * v0[26] + "NeuroPLC_Weights".w0[335] * v0[27];
    v1[12] := "NeuroPLC_Weights".w0[896 + 12] + "NeuroPLC_Weights".w0[336] * v0[0] + "NeuroPLC_Weights".w0[337] * v0[1] + "NeuroPLC_Weights".w0[338] * v0[2] + "NeuroPLC_Weights".w0[339] * v0[3] + "NeuroPLC_Weights".w0[340] * v0[4] + "NeuroPLC_Weights".w0[341] * v0[5] + "NeuroPLC_Weights".w0[342] * v0[6] + "NeuroPLC_Weights".w0[343] * v0[7] + "NeuroPLC_Weights".w0[344] * v0[8] + "NeuroPLC_Weights".w0[345] * v0[9] + "NeuroPLC_Weights".w0[346] * v0[10] + "NeuroPLC_Weights".w0[347] * v0[11] + "NeuroPLC_Weights".w0[348] * v0[12] + "NeuroPLC_Weights".w0[349] * v0[13] + "NeuroPLC_Weights".w0[350] * v0[14] + "NeuroPLC_Weights".w0[351] * v0[15] + "NeuroPLC_Weights".w0[352] * v0[16] + "NeuroPLC_Weights".w0[353] * v0[17] + "NeuroPLC_Weights".w0[354] * v0[18] + "NeuroPLC_Weights".w0[355] * v0[19] + "NeuroPLC_Weights".w0[356] * v0[20] + "NeuroPLC_Weights".w0[357] * v0[21] + "NeuroPLC_Weights".w0[358] * v0[22] + "NeuroPLC_Weights".w0[359] * v0[23] + "NeuroPLC_Weights".w0[360] * v0[24] + "NeuroPLC_Weights".w0[361] * v0[25] + "NeuroPLC_Weights".w0[362] * v0[26] + "NeuroPLC_Weights".w0[363] * v0[27];
    v1[13] := "NeuroPLC_Weights".w0[896 + 13] + "NeuroPLC_Weights".w0[364] * v0[0] + "NeuroPLC_Weights".w0[365] * v0[1] + "NeuroPLC_Weights".w0[366] * v0[2] + "NeuroPLC_Weights".w0[367] * v0[3] + "NeuroPLC_Weights".w0[368] * v0[4] + "NeuroPLC_Weights".w0[369] * v0[5] + "NeuroPLC_Weights".w0[370] * v0[6] + "NeuroPLC_Weights".w0[371] * v0[7] + "NeuroPLC_Weights".w0[372] * v0[8] + "NeuroPLC_Weights".w0[373] * v0[9] + "NeuroPLC_Weights".w0[374] * v0[10] + "NeuroPLC_Weights".w0[375] * v0[11] + "NeuroPLC_Weights".w0[376] * v0[12] + "NeuroPLC_Weights".w0[377] * v0[13] + "NeuroPLC_Weights".w0[378] * v0[14] + "NeuroPLC_Weights".w0[379] * v0[15] + "NeuroPLC_Weights".w0[380] * v0[16] + "NeuroPLC_Weights".w0[381] * v0[17] + "NeuroPLC_Weights".w0[382] * v0[18] + "NeuroPLC_Weights".w0[383] * v0[19] + "NeuroPLC_Weights".w0[384] * v0[20] + "NeuroPLC_Weights".w0[385] * v0[21] + "NeuroPLC_Weights".w0[386] * v0[22] + "NeuroPLC_Weights".w0[387] * v0[23] + "NeuroPLC_Weights".w0[388] * v0[24] + "NeuroPLC_Weights".w0[389] * v0[25] + "NeuroPLC_Weights".w0[390] * v0[26] + "NeuroPLC_Weights".w0[391] * v0[27];
    v1[14] := "NeuroPLC_Weights".w0[896 + 14] + "NeuroPLC_Weights".w0[392] * v0[0] + "NeuroPLC_Weights".w0[393] * v0[1] + "NeuroPLC_Weights".w0[394] * v0[2] + "NeuroPLC_Weights".w0[395] * v0[3] + "NeuroPLC_Weights".w0[396] * v0[4] + "NeuroPLC_Weights".w0[397] * v0[5] + "NeuroPLC_Weights".w0[398] * v0[6] + "NeuroPLC_Weights".w0[399] * v0[7] + "NeuroPLC_Weights".w0[400] * v0[8] + "NeuroPLC_Weights".w0[401] * v0[9] + "NeuroPLC_Weights".w0[402] * v0[10] + "NeuroPLC_Weights".w0[403] * v0[11] + "NeuroPLC_Weights".w0[404] * v0[12] + "NeuroPLC_Weights".w0[405] * v0[13] + "NeuroPLC_Weights".w0[406] * v0[14] + "NeuroPLC_Weights".w0[407] * v0[15] + "NeuroPLC_Weights".w0[408] * v0[16] + "NeuroPLC_Weights".w0[409] * v0[17] + "NeuroPLC_Weights".w0[410] * v0[18] + "NeuroPLC_Weights".w0[411] * v0[19] + "NeuroPLC_Weights".w0[412] * v0[20] + "NeuroPLC_Weights".w0[413] * v0[21] + "NeuroPLC_Weights".w0[414] * v0[22] + "NeuroPLC_Weights".w0[415] * v0[23] + "NeuroPLC_Weights".w0[416] * v0[24] + "NeuroPLC_Weights".w0[417] * v0[25] + "NeuroPLC_Weights".w0[418] * v0[26] + "NeuroPLC_Weights".w0[419] * v0[27];
    v1[15] := "NeuroPLC_Weights".w0[896 + 15] + "NeuroPLC_Weights".w0[420] * v0[0] + "NeuroPLC_Weights".w0[421] * v0[1] + "NeuroPLC_Weights".w0[422] * v0[2] + "NeuroPLC_Weights".w0[423] * v0[3] + "NeuroPLC_Weights".w0[424] * v0[4] + "NeuroPLC_Weights".w0[425] * v0[5] + "NeuroPLC_Weights".w0[426] * v0[6] + "NeuroPLC_Weights".w0[427] * v0[7] + "NeuroPLC_Weights".w0[428] * v0[8] + "NeuroPLC_Weights".w0[429] * v0[9] + "NeuroPLC_Weights".w0[430] * v0[10] + "NeuroPLC_Weights".w0[431] * v0[11] + "NeuroPLC_Weights".w0[432] * v0[12] + "NeuroPLC_Weights".w0[433] * v0[13] + "NeuroPLC_Weights".w0[434] * v0[14] + "NeuroPLC_Weights".w0[435] * v0[15] + "NeuroPLC_Weights".w0[436] * v0[16] + "NeuroPLC_Weights".w0[437] * v0[17] + "NeuroPLC_Weights".w0[438] * v0[18] + "NeuroPLC_Weights".w0[439] * v0[19] + "NeuroPLC_Weights".w0[440] * v0[20] + "NeuroPLC_Weights".w0[441] * v0[21] + "NeuroPLC_Weights".w0[442] * v0[22] + "NeuroPLC_Weights".w0[443] * v0[23] + "NeuroPLC_Weights".w0[444] * v0[24] + "NeuroPLC_Weights".w0[445] * v0[25] + "NeuroPLC_Weights".w0[446] * v0[26] + "NeuroPLC_Weights".w0[447] * v0[27];
    v1[16] := "NeuroPLC_Weights".w0[896 + 16] + "NeuroPLC_Weights".w0[448] * v0[0] + "NeuroPLC_Weights".w0[449] * v0[1] + "NeuroPLC_Weights".w0[450] * v0[2] + "NeuroPLC_Weights".w0[451] * v0[3] + "NeuroPLC_Weights".w0[452] * v0[4] + "NeuroPLC_Weights".w0[453] * v0[5] + "NeuroPLC_Weights".w0[454] * v0[6] + "NeuroPLC_Weights".w0[455] * v0[7] + "NeuroPLC_Weights".w0[456] * v0[8] + "NeuroPLC_Weights".w0[457] * v0[9] + "NeuroPLC_Weights".w0[458] * v0[10] + "NeuroPLC_Weights".w0[459] * v0[11] + "NeuroPLC_Weights".w0[460] * v0[12] + "NeuroPLC_Weights".w0[461] * v0[13] + "NeuroPLC_Weights".w0[462] * v0[14] + "NeuroPLC_Weights".w0[463] * v0[15] + "NeuroPLC_Weights".w0[464] * v0[16] + "NeuroPLC_Weights".w0[465] * v0[17] + "NeuroPLC_Weights".w0[466] * v0[18] + "NeuroPLC_Weights".w0[467] * v0[19] + "NeuroPLC_Weights".w0[468] * v0[20] + "NeuroPLC_Weights".w0[469] * v0[21] + "NeuroPLC_Weights".w0[470] * v0[22] + "NeuroPLC_Weights".w0[471] * v0[23] + "NeuroPLC_Weights".w0[472] * v0[24] + "NeuroPLC_Weights".w0[473] * v0[25] + "NeuroPLC_Weights".w0[474] * v0[26] + "NeuroPLC_Weights".w0[475] * v0[27];
    v1[17] := "NeuroPLC_Weights".w0[896 + 17] + "NeuroPLC_Weights".w0[476] * v0[0] + "NeuroPLC_Weights".w0[477] * v0[1] + "NeuroPLC_Weights".w0[478] * v0[2] + "NeuroPLC_Weights".w0[479] * v0[3] + "NeuroPLC_Weights".w0[480] * v0[4] + "NeuroPLC_Weights".w0[481] * v0[5] + "NeuroPLC_Weights".w0[482] * v0[6] + "NeuroPLC_Weights".w0[483] * v0[7] + "NeuroPLC_Weights".w0[484] * v0[8] + "NeuroPLC_Weights".w0[485] * v0[9] + "NeuroPLC_Weights".w0[486] * v0[10] + "NeuroPLC_Weights".w0[487] * v0[11] + "NeuroPLC_Weights".w0[488] * v0[12] + "NeuroPLC_Weights".w0[489] * v0[13] + "NeuroPLC_Weights".w0[490] * v0[14] + "NeuroPLC_Weights".w0[491] * v0[15] + "NeuroPLC_Weights".w0[492] * v0[16] + "NeuroPLC_Weights".w0[493] * v0[17] + "NeuroPLC_Weights".w0[494] * v0[18] + "NeuroPLC_Weights".w0[495] * v0[19] + "NeuroPLC_Weights".w0[496] * v0[20] + "NeuroPLC_Weights".w0[497] * v0[21] + "NeuroPLC_Weights".w0[498] * v0[22] + "NeuroPLC_Weights".w0[499] * v0[23] + "NeuroPLC_Weights".w0[500] * v0[24] + "NeuroPLC_Weights".w0[501] * v0[25] + "NeuroPLC_Weights".w0[502] * v0[26] + "NeuroPLC_Weights".w0[503] * v0[27];
    v1[18] := "NeuroPLC_Weights".w0[896 + 18] + "NeuroPLC_Weights".w0[504] * v0[0] + "NeuroPLC_Weights".w0[505] * v0[1] + "NeuroPLC_Weights".w0[506] * v0[2] + "NeuroPLC_Weights".w0[507] * v0[3] + "NeuroPLC_Weights".w0[508] * v0[4] + "NeuroPLC_Weights".w0[509] * v0[5] + "NeuroPLC_Weights".w0[510] * v0[6] + "NeuroPLC_Weights".w0[511] * v0[7] + "NeuroPLC_Weights".w0[512] * v0[8] + "NeuroPLC_Weights".w0[513] * v0[9] + "NeuroPLC_Weights".w0[514] * v0[10] + "NeuroPLC_Weights".w0[515] * v0[11] + "NeuroPLC_Weights".w0[516] * v0[12] + "NeuroPLC_Weights".w0[517] * v0[13] + "NeuroPLC_Weights".w0[518] * v0[14] + "NeuroPLC_Weights".w0[519] * v0[15] + "NeuroPLC_Weights".w0[520] * v0[16] + "NeuroPLC_Weights".w0[521] * v0[17] + "NeuroPLC_Weights".w0[522] * v0[18] + "NeuroPLC_Weights".w0[523] * v0[19] + "NeuroPLC_Weights".w0[524] * v0[20] + "NeuroPLC_Weights".w0[525] * v0[21] + "NeuroPLC_Weights".w0[526] * v0[22] + "NeuroPLC_Weights".w0[527] * v0[23] + "NeuroPLC_Weights".w0[528] * v0[24] + "NeuroPLC_Weights".w0[529] * v0[25] + "NeuroPLC_Weights".w0[530] * v0[26] + "NeuroPLC_Weights".w0[531] * v0[27];
    v1[19] := "NeuroPLC_Weights".w0[896 + 19] + "NeuroPLC_Weights".w0[532] * v0[0] + "NeuroPLC_Weights".w0[533] * v0[1] + "NeuroPLC_Weights".w0[534] * v0[2] + "NeuroPLC_Weights".w0[535] * v0[3] + "NeuroPLC_Weights".w0[536] * v0[4] + "NeuroPLC_Weights".w0[537] * v0[5] + "NeuroPLC_Weights".w0[538] * v0[6] + "NeuroPLC_Weights".w0[539] * v0[7] + "NeuroPLC_Weights".w0[540] * v0[8] + "NeuroPLC_Weights".w0[541] * v0[9] + "NeuroPLC_Weights".w0[542] * v0[10] + "NeuroPLC_Weights".w0[543] * v0[11] + "NeuroPLC_Weights".w0[544] * v0[12] + "NeuroPLC_Weights".w0[545] * v0[13] + "NeuroPLC_Weights".w0[546] * v0[14] + "NeuroPLC_Weights".w0[547] * v0[15] + "NeuroPLC_Weights".w0[548] * v0[16] + "NeuroPLC_Weights".w0[549] * v0[17] + "NeuroPLC_Weights".w0[550] * v0[18] + "NeuroPLC_Weights".w0[551] * v0[19] + "NeuroPLC_Weights".w0[552] * v0[20] + "NeuroPLC_Weights".w0[553] * v0[21] + "NeuroPLC_Weights".w0[554] * v0[22] + "NeuroPLC_Weights".w0[555] * v0[23] + "NeuroPLC_Weights".w0[556] * v0[24] + "NeuroPLC_Weights".w0[557] * v0[25] + "NeuroPLC_Weights".w0[558] * v0[26] + "NeuroPLC_Weights".w0[559] * v0[27];
    v1[20] := "NeuroPLC_Weights".w0[896 + 20] + "NeuroPLC_Weights".w0[560] * v0[0] + "NeuroPLC_Weights".w0[561] * v0[1] + "NeuroPLC_Weights".w0[562] * v0[2] + "NeuroPLC_Weights".w0[563] * v0[3] + "NeuroPLC_Weights".w0[564] * v0[4] + "NeuroPLC_Weights".w0[565] * v0[5] + "NeuroPLC_Weights".w0[566] * v0[6] + "NeuroPLC_Weights".w0[567] * v0[7] + "NeuroPLC_Weights".w0[568] * v0[8] + "NeuroPLC_Weights".w0[569] * v0[9] + "NeuroPLC_Weights".w0[570] * v0[10] + "NeuroPLC_Weights".w0[571] * v0[11] + "NeuroPLC_Weights".w0[572] * v0[12] + "NeuroPLC_Weights".w0[573] * v0[13] + "NeuroPLC_Weights".w0[574] * v0[14] + "NeuroPLC_Weights".w0[575] * v0[15] + "NeuroPLC_Weights".w0[576] * v0[16] + "NeuroPLC_Weights".w0[577] * v0[17] + "NeuroPLC_Weights".w0[578] * v0[18] + "NeuroPLC_Weights".w0[579] * v0[19] + "NeuroPLC_Weights".w0[580] * v0[20] + "NeuroPLC_Weights".w0[581] * v0[21] + "NeuroPLC_Weights".w0[582] * v0[22] + "NeuroPLC_Weights".w0[583] * v0[23] + "NeuroPLC_Weights".w0[584] * v0[24] + "NeuroPLC_Weights".w0[585] * v0[25] + "NeuroPLC_Weights".w0[586] * v0[26] + "NeuroPLC_Weights".w0[587] * v0[27];
    v1[21] := "NeuroPLC_Weights".w0[896 + 21] + "NeuroPLC_Weights".w0[588] * v0[0] + "NeuroPLC_Weights".w0[589] * v0[1] + "NeuroPLC_Weights".w0[590] * v0[2] + "NeuroPLC_Weights".w0[591] * v0[3] + "NeuroPLC_Weights".w0[592] * v0[4] + "NeuroPLC_Weights".w0[593] * v0[5] + "NeuroPLC_Weights".w0[594] * v0[6] + "NeuroPLC_Weights".w0[595] * v0[7] + "NeuroPLC_Weights".w0[596] * v0[8] + "NeuroPLC_Weights".w0[597] * v0[9] + "NeuroPLC_Weights".w0[598] * v0[10] + "NeuroPLC_Weights".w0[599] * v0[11] + "NeuroPLC_Weights".w0[600] * v0[12] + "NeuroPLC_Weights".w0[601] * v0[13] + "NeuroPLC_Weights".w0[602] * v0[14] + "NeuroPLC_Weights".w0[603] * v0[15] + "NeuroPLC_Weights".w0[604] * v0[16] + "NeuroPLC_Weights".w0[605] * v0[17] + "NeuroPLC_Weights".w0[606] * v0[18] + "NeuroPLC_Weights".w0[607] * v0[19] + "NeuroPLC_Weights".w0[608] * v0[20] + "NeuroPLC_Weights".w0[609] * v0[21] + "NeuroPLC_Weights".w0[610] * v0[22] + "NeuroPLC_Weights".w0[611] * v0[23] + "NeuroPLC_Weights".w0[612] * v0[24] + "NeuroPLC_Weights".w0[613] * v0[25] + "NeuroPLC_Weights".w0[614] * v0[26] + "NeuroPLC_Weights".w0[615] * v0[27];
    v1[22] := "NeuroPLC_Weights".w0[896 + 22] + "NeuroPLC_Weights".w0[616] * v0[0] + "NeuroPLC_Weights".w0[617] * v0[1] + "NeuroPLC_Weights".w0[618] * v0[2] + "NeuroPLC_Weights".w0[619] * v0[3] + "NeuroPLC_Weights".w0[620] * v0[4] + "NeuroPLC_Weights".w0[621] * v0[5] + "NeuroPLC_Weights".w0[622] * v0[6] + "NeuroPLC_Weights".w0[623] * v0[7] + "NeuroPLC_Weights".w0[624] * v0[8] + "NeuroPLC_Weights".w0[625] * v0[9] + "NeuroPLC_Weights".w0[626] * v0[10] + "NeuroPLC_Weights".w0[627] * v0[11] + "NeuroPLC_Weights".w0[628] * v0[12] + "NeuroPLC_Weights".w0[629] * v0[13] + "NeuroPLC_Weights".w0[630] * v0[14] + "NeuroPLC_Weights".w0[631] * v0[15] + "NeuroPLC_Weights".w0[632] * v0[16] + "NeuroPLC_Weights".w0[633] * v0[17] + "NeuroPLC_Weights".w0[634] * v0[18] + "NeuroPLC_Weights".w0[635] * v0[19] + "NeuroPLC_Weights".w0[636] * v0[20] + "NeuroPLC_Weights".w0[637] * v0[21] + "NeuroPLC_Weights".w0[638] * v0[22] + "NeuroPLC_Weights".w0[639] * v0[23] + "NeuroPLC_Weights".w0[640] * v0[24] + "NeuroPLC_Weights".w0[641] * v0[25] + "NeuroPLC_Weights".w0[642] * v0[26] + "NeuroPLC_Weights".w0[643] * v0[27];
    v1[23] := "NeuroPLC_Weights".w0[896 + 23] + "NeuroPLC_Weights".w0[644] * v0[0] + "NeuroPLC_Weights".w0[645] * v0[1] + "NeuroPLC_Weights".w0[646] * v0[2] + "NeuroPLC_Weights".w0[647] * v0[3] + "NeuroPLC_Weights".w0[648] * v0[4] + "NeuroPLC_Weights".w0[649] * v0[5] + "NeuroPLC_Weights".w0[650] * v0[6] + "NeuroPLC_Weights".w0[651] * v0[7] + "NeuroPLC_Weights".w0[652] * v0[8] + "NeuroPLC_Weights".w0[653] * v0[9] + "NeuroPLC_Weights".w0[654] * v0[10] + "NeuroPLC_Weights".w0[655] * v0[11] + "NeuroPLC_Weights".w0[656] * v0[12] + "NeuroPLC_Weights".w0[657] * v0[13] + "NeuroPLC_Weights".w0[658] * v0[14] + "NeuroPLC_Weights".w0[659] * v0[15] + "NeuroPLC_Weights".w0[660] * v0[16] + "NeuroPLC_Weights".w0[661] * v0[17] + "NeuroPLC_Weights".w0[662] * v0[18] + "NeuroPLC_Weights".w0[663] * v0[19] + "NeuroPLC_Weights".w0[664] * v0[20] + "NeuroPLC_Weights".w0[665] * v0[21] + "NeuroPLC_Weights".w0[666] * v0[22] + "NeuroPLC_Weights".w0[667] * v0[23] + "NeuroPLC_Weights".w0[668] * v0[24] + "NeuroPLC_Weights".w0[669] * v0[25] + "NeuroPLC_Weights".w0[670] * v0[26] + "NeuroPLC_Weights".w0[671] * v0[27];
    v1[24] := "NeuroPLC_Weights".w0[896 + 24] + "NeuroPLC_Weights".w0[672] * v0[0] + "NeuroPLC_Weights".w0[673] * v0[1] + "NeuroPLC_Weights".w0[674] * v0[2] + "NeuroPLC_Weights".w0[675] * v0[3] + "NeuroPLC_Weights".w0[676] * v0[4] + "NeuroPLC_Weights".w0[677] * v0[5] + "NeuroPLC_Weights".w0[678] * v0[6] + "NeuroPLC_Weights".w0[679] * v0[7] + "NeuroPLC_Weights".w0[680] * v0[8] + "NeuroPLC_Weights".w0[681] * v0[9] + "NeuroPLC_Weights".w0[682] * v0[10] + "NeuroPLC_Weights".w0[683] * v0[11] + "NeuroPLC_Weights".w0[684] * v0[12] + "NeuroPLC_Weights".w0[685] * v0[13] + "NeuroPLC_Weights".w0[686] * v0[14] + "NeuroPLC_Weights".w0[687] * v0[15] + "NeuroPLC_Weights".w0[688] * v0[16] + "NeuroPLC_Weights".w0[689] * v0[17] + "NeuroPLC_Weights".w0[690] * v0[18] + "NeuroPLC_Weights".w0[691] * v0[19] + "NeuroPLC_Weights".w0[692] * v0[20] + "NeuroPLC_Weights".w0[693] * v0[21] + "NeuroPLC_Weights".w0[694] * v0[22] + "NeuroPLC_Weights".w0[695] * v0[23] + "NeuroPLC_Weights".w0[696] * v0[24] + "NeuroPLC_Weights".w0[697] * v0[25] + "NeuroPLC_Weights".w0[698] * v0[26] + "NeuroPLC_Weights".w0[699] * v0[27];
    v1[25] := "NeuroPLC_Weights".w0[896 + 25] + "NeuroPLC_Weights".w0[700] * v0[0] + "NeuroPLC_Weights".w0[701] * v0[1] + "NeuroPLC_Weights".w0[702] * v0[2] + "NeuroPLC_Weights".w0[703] * v0[3] + "NeuroPLC_Weights".w0[704] * v0[4] + "NeuroPLC_Weights".w0[705] * v0[5] + "NeuroPLC_Weights".w0[706] * v0[6] + "NeuroPLC_Weights".w0[707] * v0[7] + "NeuroPLC_Weights".w0[708] * v0[8] + "NeuroPLC_Weights".w0[709] * v0[9] + "NeuroPLC_Weights".w0[710] * v0[10] + "NeuroPLC_Weights".w0[711] * v0[11] + "NeuroPLC_Weights".w0[712] * v0[12] + "NeuroPLC_Weights".w0[713] * v0[13] + "NeuroPLC_Weights".w0[714] * v0[14] + "NeuroPLC_Weights".w0[715] * v0[15] + "NeuroPLC_Weights".w0[716] * v0[16] + "NeuroPLC_Weights".w0[717] * v0[17] + "NeuroPLC_Weights".w0[718] * v0[18] + "NeuroPLC_Weights".w0[719] * v0[19] + "NeuroPLC_Weights".w0[720] * v0[20] + "NeuroPLC_Weights".w0[721] * v0[21] + "NeuroPLC_Weights".w0[722] * v0[22] + "NeuroPLC_Weights".w0[723] * v0[23] + "NeuroPLC_Weights".w0[724] * v0[24] + "NeuroPLC_Weights".w0[725] * v0[25] + "NeuroPLC_Weights".w0[726] * v0[26] + "NeuroPLC_Weights".w0[727] * v0[27];
    v1[26] := "NeuroPLC_Weights".w0[896 + 26] + "NeuroPLC_Weights".w0[728] * v0[0] + "NeuroPLC_Weights".w0[729] * v0[1] + "NeuroPLC_Weights".w0[730] * v0[2] + "NeuroPLC_Weights".w0[731] * v0[3] + "NeuroPLC_Weights".w0[732] * v0[4] + "NeuroPLC_Weights".w0[733] * v0[5] + "NeuroPLC_Weights".w0[734] * v0[6] + "NeuroPLC_Weights".w0[735] * v0[7] + "NeuroPLC_Weights".w0[736] * v0[8] + "NeuroPLC_Weights".w0[737] * v0[9] + "NeuroPLC_Weights".w0[738] * v0[10] + "NeuroPLC_Weights".w0[739] * v0[11] + "NeuroPLC_Weights".w0[740] * v0[12] + "NeuroPLC_Weights".w0[741] * v0[13] + "NeuroPLC_Weights".w0[742] * v0[14] + "NeuroPLC_Weights".w0[743] * v0[15] + "NeuroPLC_Weights".w0[744] * v0[16] + "NeuroPLC_Weights".w0[745] * v0[17] + "NeuroPLC_Weights".w0[746] * v0[18] + "NeuroPLC_Weights".w0[747] * v0[19] + "NeuroPLC_Weights".w0[748] * v0[20] + "NeuroPLC_Weights".w0[749] * v0[21] + "NeuroPLC_Weights".w0[750] * v0[22] + "NeuroPLC_Weights".w0[751] * v0[23] + "NeuroPLC_Weights".w0[752] * v0[24] + "NeuroPLC_Weights".w0[753] * v0[25] + "NeuroPLC_Weights".w0[754] * v0[26] + "NeuroPLC_Weights".w0[755] * v0[27];
    v1[27] := "NeuroPLC_Weights".w0[896 + 27] + "NeuroPLC_Weights".w0[756] * v0[0] + "NeuroPLC_Weights".w0[757] * v0[1] + "NeuroPLC_Weights".w0[758] * v0[2] + "NeuroPLC_Weights".w0[759] * v0[3] + "NeuroPLC_Weights".w0[760] * v0[4] + "NeuroPLC_Weights".w0[761] * v0[5] + "NeuroPLC_Weights".w0[762] * v0[6] + "NeuroPLC_Weights".w0[763] * v0[7] + "NeuroPLC_Weights".w0[764] * v0[8] + "NeuroPLC_Weights".w0[765] * v0[9] + "NeuroPLC_Weights".w0[766] * v0[10] + "NeuroPLC_Weights".w0[767] * v0[11] + "NeuroPLC_Weights".w0[768] * v0[12] + "NeuroPLC_Weights".w0[769] * v0[13] + "NeuroPLC_Weights".w0[770] * v0[14] + "NeuroPLC_Weights".w0[771] * v0[15] + "NeuroPLC_Weights".w0[772] * v0[16] + "NeuroPLC_Weights".w0[773] * v0[17] + "NeuroPLC_Weights".w0[774] * v0[18] + "NeuroPLC_Weights".w0[775] * v0[19] + "NeuroPLC_Weights".w0[776] * v0[20] + "NeuroPLC_Weights".w0[777] * v0[21] + "NeuroPLC_Weights".w0[778] * v0[22] + "NeuroPLC_Weights".w0[779] * v0[23] + "NeuroPLC_Weights".w0[780] * v0[24] + "NeuroPLC_Weights".w0[781] * v0[25] + "NeuroPLC_Weights".w0[782] * v0[26] + "NeuroPLC_Weights".w0[783] * v0[27];
    v1[28] := "NeuroPLC_Weights".w0[896 + 28] + "NeuroPLC_Weights".w0[784] * v0[0] + "NeuroPLC_Weights".w0[785] * v0[1] + "NeuroPLC_Weights".w0[786] * v0[2] + "NeuroPLC_Weights".w0[787] * v0[3] + "NeuroPLC_Weights".w0[788] * v0[4] + "NeuroPLC_Weights".w0[789] * v0[5] + "NeuroPLC_Weights".w0[790] * v0[6] + "NeuroPLC_Weights".w0[791] * v0[7] + "NeuroPLC_Weights".w0[792] * v0[8] + "NeuroPLC_Weights".w0[793] * v0[9] + "NeuroPLC_Weights".w0[794] * v0[10] + "NeuroPLC_Weights".w0[795] * v0[11] + "NeuroPLC_Weights".w0[796] * v0[12] + "NeuroPLC_Weights".w0[797] * v0[13] + "NeuroPLC_Weights".w0[798] * v0[14] + "NeuroPLC_Weights".w0[799] * v0[15] + "NeuroPLC_Weights".w0[800] * v0[16] + "NeuroPLC_Weights".w0[801] * v0[17] + "NeuroPLC_Weights".w0[802] * v0[18] + "NeuroPLC_Weights".w0[803] * v0[19] + "NeuroPLC_Weights".w0[804] * v0[20] + "NeuroPLC_Weights".w0[805] * v0[21] + "NeuroPLC_Weights".w0[806] * v0[22] + "NeuroPLC_Weights".w0[807] * v0[23] + "NeuroPLC_Weights".w0[808] * v0[24] + "NeuroPLC_Weights".w0[809] * v0[25] + "NeuroPLC_Weights".w0[810] * v0[26] + "NeuroPLC_Weights".w0[811] * v0[27];
    v1[29] := "NeuroPLC_Weights".w0[896 + 29] + "NeuroPLC_Weights".w0[812] * v0[0] + "NeuroPLC_Weights".w0[813] * v0[1] + "NeuroPLC_Weights".w0[814] * v0[2] + "NeuroPLC_Weights".w0[815] * v0[3] + "NeuroPLC_Weights".w0[816] * v0[4] + "NeuroPLC_Weights".w0[817] * v0[5] + "NeuroPLC_Weights".w0[818] * v0[6] + "NeuroPLC_Weights".w0[819] * v0[7] + "NeuroPLC_Weights".w0[820] * v0[8] + "NeuroPLC_Weights".w0[821] * v0[9] + "NeuroPLC_Weights".w0[822] * v0[10] + "NeuroPLC_Weights".w0[823] * v0[11] + "NeuroPLC_Weights".w0[824] * v0[12] + "NeuroPLC_Weights".w0[825] * v0[13] + "NeuroPLC_Weights".w0[826] * v0[14] + "NeuroPLC_Weights".w0[827] * v0[15] + "NeuroPLC_Weights".w0[828] * v0[16] + "NeuroPLC_Weights".w0[829] * v0[17] + "NeuroPLC_Weights".w0[830] * v0[18] + "NeuroPLC_Weights".w0[831] * v0[19] + "NeuroPLC_Weights".w0[832] * v0[20] + "NeuroPLC_Weights".w0[833] * v0[21] + "NeuroPLC_Weights".w0[834] * v0[22] + "NeuroPLC_Weights".w0[835] * v0[23] + "NeuroPLC_Weights".w0[836] * v0[24] + "NeuroPLC_Weights".w0[837] * v0[25] + "NeuroPLC_Weights".w0[838] * v0[26] + "NeuroPLC_Weights".w0[839] * v0[27];
    v1[30] := "NeuroPLC_Weights".w0[896 + 30] + "NeuroPLC_Weights".w0[840] * v0[0] + "NeuroPLC_Weights".w0[841] * v0[1] + "NeuroPLC_Weights".w0[842] * v0[2] + "NeuroPLC_Weights".w0[843] * v0[3] + "NeuroPLC_Weights".w0[844] * v0[4] + "NeuroPLC_Weights".w0[845] * v0[5] + "NeuroPLC_Weights".w0[846] * v0[6] + "NeuroPLC_Weights".w0[847] * v0[7] + "NeuroPLC_Weights".w0[848] * v0[8] + "NeuroPLC_Weights".w0[849] * v0[9] + "NeuroPLC_Weights".w0[850] * v0[10] + "NeuroPLC_Weights".w0[851] * v0[11] + "NeuroPLC_Weights".w0[852] * v0[12] + "NeuroPLC_Weights".w0[853] * v0[13] + "NeuroPLC_Weights".w0[854] * v0[14] + "NeuroPLC_Weights".w0[855] * v0[15] + "NeuroPLC_Weights".w0[856] * v0[16] + "NeuroPLC_Weights".w0[857] * v0[17] + "NeuroPLC_Weights".w0[858] * v0[18] + "NeuroPLC_Weights".w0[859] * v0[19] + "NeuroPLC_Weights".w0[860] * v0[20] + "NeuroPLC_Weights".w0[861] * v0[21] + "NeuroPLC_Weights".w0[862] * v0[22] + "NeuroPLC_Weights".w0[863] * v0[23] + "NeuroPLC_Weights".w0[864] * v0[24] + "NeuroPLC_Weights".w0[865] * v0[25] + "NeuroPLC_Weights".w0[866] * v0[26] + "NeuroPLC_Weights".w0[867] * v0[27];
    v1[31] := "NeuroPLC_Weights".w0[896 + 31] + "NeuroPLC_Weights".w0[868] * v0[0] + "NeuroPLC_Weights".w0[869] * v0[1] + "NeuroPLC_Weights".w0[870] * v0[2] + "NeuroPLC_Weights".w0[871] * v0[3] + "NeuroPLC_Weights".w0[872] * v0[4] + "NeuroPLC_Weights".w0[873] * v0[5] + "NeuroPLC_Weights".w0[874] * v0[6] + "NeuroPLC_Weights".w0[875] * v0[7] + "NeuroPLC_Weights".w0[876] * v0[8] + "NeuroPLC_Weights".w0[877] * v0[9] + "NeuroPLC_Weights".w0[878] * v0[10] + "NeuroPLC_Weights".w0[879] * v0[11] + "NeuroPLC_Weights".w0[880] * v0[12] + "NeuroPLC_Weights".w0[881] * v0[13] + "NeuroPLC_Weights".w0[882] * v0[14] + "NeuroPLC_Weights".w0[883] * v0[15] + "NeuroPLC_Weights".w0[884] * v0[16] + "NeuroPLC_Weights".w0[885] * v0[17] + "NeuroPLC_Weights".w0[886] * v0[18] + "NeuroPLC_Weights".w0[887] * v0[19] + "NeuroPLC_Weights".w0[888] * v0[20] + "NeuroPLC_Weights".w0[889] * v0[21] + "NeuroPLC_Weights".w0[890] * v0[22] + "NeuroPLC_Weights".w0[891] * v0[23] + "NeuroPLC_Weights".w0[892] * v0[24] + "NeuroPLC_Weights".w0[893] * v0[25] + "NeuroPLC_Weights".w0[894] * v0[26] + "NeuroPLC_Weights".w0[895] * v0[27];

    // ---- relu0: RELU ----
    IF v1[0] > 0.0 THEN v2[0] := v1[0]; ELSE v2[0] := 0.0; END_IF;
    IF v1[1] > 0.0 THEN v2[1] := v1[1]; ELSE v2[1] := 0.0; END_IF;
    IF v1[2] > 0.0 THEN v2[2] := v1[2]; ELSE v2[2] := 0.0; END_IF;
    IF v1[3] > 0.0 THEN v2[3] := v1[3]; ELSE v2[3] := 0.0; END_IF;
    IF v1[4] > 0.0 THEN v2[4] := v1[4]; ELSE v2[4] := 0.0; END_IF;
    IF v1[5] > 0.0 THEN v2[5] := v1[5]; ELSE v2[5] := 0.0; END_IF;
    IF v1[6] > 0.0 THEN v2[6] := v1[6]; ELSE v2[6] := 0.0; END_IF;
    IF v1[7] > 0.0 THEN v2[7] := v1[7]; ELSE v2[7] := 0.0; END_IF;
    IF v1[8] > 0.0 THEN v2[8] := v1[8]; ELSE v2[8] := 0.0; END_IF;
    IF v1[9] > 0.0 THEN v2[9] := v1[9]; ELSE v2[9] := 0.0; END_IF;
    IF v1[10] > 0.0 THEN v2[10] := v1[10]; ELSE v2[10] := 0.0; END_IF;
    IF v1[11] > 0.0 THEN v2[11] := v1[11]; ELSE v2[11] := 0.0; END_IF;
    IF v1[12] > 0.0 THEN v2[12] := v1[12]; ELSE v2[12] := 0.0; END_IF;
    IF v1[13] > 0.0 THEN v2[13] := v1[13]; ELSE v2[13] := 0.0; END_IF;
    IF v1[14] > 0.0 THEN v2[14] := v1[14]; ELSE v2[14] := 0.0; END_IF;
    IF v1[15] > 0.0 THEN v2[15] := v1[15]; ELSE v2[15] := 0.0; END_IF;
    IF v1[16] > 0.0 THEN v2[16] := v1[16]; ELSE v2[16] := 0.0; END_IF;
    IF v1[17] > 0.0 THEN v2[17] := v1[17]; ELSE v2[17] := 0.0; END_IF;
    IF v1[18] > 0.0 THEN v2[18] := v1[18]; ELSE v2[18] := 0.0; END_IF;
    IF v1[19] > 0.0 THEN v2[19] := v1[19]; ELSE v2[19] := 0.0; END_IF;
    IF v1[20] > 0.0 THEN v2[20] := v1[20]; ELSE v2[20] := 0.0; END_IF;
    IF v1[21] > 0.0 THEN v2[21] := v1[21]; ELSE v2[21] := 0.0; END_IF;
    IF v1[22] > 0.0 THEN v2[22] := v1[22]; ELSE v2[22] := 0.0; END_IF;
    IF v1[23] > 0.0 THEN v2[23] := v1[23]; ELSE v2[23] := 0.0; END_IF;
    IF v1[24] > 0.0 THEN v2[24] := v1[24]; ELSE v2[24] := 0.0; END_IF;
    IF v1[25] > 0.0 THEN v2[25] := v1[25]; ELSE v2[25] := 0.0; END_IF;
    IF v1[26] > 0.0 THEN v2[26] := v1[26]; ELSE v2[26] := 0.0; END_IF;
    IF v1[27] > 0.0 THEN v2[27] := v1[27]; ELSE v2[27] := 0.0; END_IF;
    IF v1[28] > 0.0 THEN v2[28] := v1[28]; ELSE v2[28] := 0.0; END_IF;
    IF v1[29] > 0.0 THEN v2[29] := v1[29]; ELSE v2[29] := 0.0; END_IF;
    IF v1[30] > 0.0 THEN v2[30] := v1[30]; ELSE v2[30] := 0.0; END_IF;
    IF v1[31] > 0.0 THEN v2[31] := v1[31]; ELSE v2[31] := 0.0; END_IF;

    // ---- fc1: MatMul(32→16) ----
    // W = "NeuroPLC_Weights".w1[:512],   b = w1[512:]
    v3[0] := "NeuroPLC_Weights".w1[512 + 0] + "NeuroPLC_Weights".w1[0] * v2[0] + "NeuroPLC_Weights".w1[1] * v2[1] + "NeuroPLC_Weights".w1[2] * v2[2] + "NeuroPLC_Weights".w1[3] * v2[3] + "NeuroPLC_Weights".w1[4] * v2[4] + "NeuroPLC_Weights".w1[5] * v2[5] + "NeuroPLC_Weights".w1[6] * v2[6] + "NeuroPLC_Weights".w1[7] * v2[7] + "NeuroPLC_Weights".w1[8] * v2[8] + "NeuroPLC_Weights".w1[9] * v2[9] + "NeuroPLC_Weights".w1[10] * v2[10] + "NeuroPLC_Weights".w1[11] * v2[11] + "NeuroPLC_Weights".w1[12] * v2[12] + "NeuroPLC_Weights".w1[13] * v2[13] + "NeuroPLC_Weights".w1[14] * v2[14] + "NeuroPLC_Weights".w1[15] * v2[15] + "NeuroPLC_Weights".w1[16] * v2[16] + "NeuroPLC_Weights".w1[17] * v2[17] + "NeuroPLC_Weights".w1[18] * v2[18] + "NeuroPLC_Weights".w1[19] * v2[19] + "NeuroPLC_Weights".w1[20] * v2[20] + "NeuroPLC_Weights".w1[21] * v2[21] + "NeuroPLC_Weights".w1[22] * v2[22] + "NeuroPLC_Weights".w1[23] * v2[23] + "NeuroPLC_Weights".w1[24] * v2[24] + "NeuroPLC_Weights".w1[25] * v2[25] + "NeuroPLC_Weights".w1[26] * v2[26] + "NeuroPLC_Weights".w1[27] * v2[27] + "NeuroPLC_Weights".w1[28] * v2[28] + "NeuroPLC_Weights".w1[29] * v2[29] + "NeuroPLC_Weights".w1[30] * v2[30] + "NeuroPLC_Weights".w1[31] * v2[31];
    v3[1] := "NeuroPLC_Weights".w1[512 + 1] + "NeuroPLC_Weights".w1[32] * v2[0] + "NeuroPLC_Weights".w1[33] * v2[1] + "NeuroPLC_Weights".w1[34] * v2[2] + "NeuroPLC_Weights".w1[35] * v2[3] + "NeuroPLC_Weights".w1[36] * v2[4] + "NeuroPLC_Weights".w1[37] * v2[5] + "NeuroPLC_Weights".w1[38] * v2[6] + "NeuroPLC_Weights".w1[39] * v2[7] + "NeuroPLC_Weights".w1[40] * v2[8] + "NeuroPLC_Weights".w1[41] * v2[9] + "NeuroPLC_Weights".w1[42] * v2[10] + "NeuroPLC_Weights".w1[43] * v2[11] + "NeuroPLC_Weights".w1[44] * v2[12] + "NeuroPLC_Weights".w1[45] * v2[13] + "NeuroPLC_Weights".w1[46] * v2[14] + "NeuroPLC_Weights".w1[47] * v2[15] + "NeuroPLC_Weights".w1[48] * v2[16] + "NeuroPLC_Weights".w1[49] * v2[17] + "NeuroPLC_Weights".w1[50] * v2[18] + "NeuroPLC_Weights".w1[51] * v2[19] + "NeuroPLC_Weights".w1[52] * v2[20] + "NeuroPLC_Weights".w1[53] * v2[21] + "NeuroPLC_Weights".w1[54] * v2[22] + "NeuroPLC_Weights".w1[55] * v2[23] + "NeuroPLC_Weights".w1[56] * v2[24] + "NeuroPLC_Weights".w1[57] * v2[25] + "NeuroPLC_Weights".w1[58] * v2[26] + "NeuroPLC_Weights".w1[59] * v2[27] + "NeuroPLC_Weights".w1[60] * v2[28] + "NeuroPLC_Weights".w1[61] * v2[29] + "NeuroPLC_Weights".w1[62] * v2[30] + "NeuroPLC_Weights".w1[63] * v2[31];
    v3[2] := "NeuroPLC_Weights".w1[512 + 2] + "NeuroPLC_Weights".w1[64] * v2[0] + "NeuroPLC_Weights".w1[65] * v2[1] + "NeuroPLC_Weights".w1[66] * v2[2] + "NeuroPLC_Weights".w1[67] * v2[3] + "NeuroPLC_Weights".w1[68] * v2[4] + "NeuroPLC_Weights".w1[69] * v2[5] + "NeuroPLC_Weights".w1[70] * v2[6] + "NeuroPLC_Weights".w1[71] * v2[7] + "NeuroPLC_Weights".w1[72] * v2[8] + "NeuroPLC_Weights".w1[73] * v2[9] + "NeuroPLC_Weights".w1[74] * v2[10] + "NeuroPLC_Weights".w1[75] * v2[11] + "NeuroPLC_Weights".w1[76] * v2[12] + "NeuroPLC_Weights".w1[77] * v2[13] + "NeuroPLC_Weights".w1[78] * v2[14] + "NeuroPLC_Weights".w1[79] * v2[15] + "NeuroPLC_Weights".w1[80] * v2[16] + "NeuroPLC_Weights".w1[81] * v2[17] + "NeuroPLC_Weights".w1[82] * v2[18] + "NeuroPLC_Weights".w1[83] * v2[19] + "NeuroPLC_Weights".w1[84] * v2[20] + "NeuroPLC_Weights".w1[85] * v2[21] + "NeuroPLC_Weights".w1[86] * v2[22] + "NeuroPLC_Weights".w1[87] * v2[23] + "NeuroPLC_Weights".w1[88] * v2[24] + "NeuroPLC_Weights".w1[89] * v2[25] + "NeuroPLC_Weights".w1[90] * v2[26] + "NeuroPLC_Weights".w1[91] * v2[27] + "NeuroPLC_Weights".w1[92] * v2[28] + "NeuroPLC_Weights".w1[93] * v2[29] + "NeuroPLC_Weights".w1[94] * v2[30] + "NeuroPLC_Weights".w1[95] * v2[31];
    v3[3] := "NeuroPLC_Weights".w1[512 + 3] + "NeuroPLC_Weights".w1[96] * v2[0] + "NeuroPLC_Weights".w1[97] * v2[1] + "NeuroPLC_Weights".w1[98] * v2[2] + "NeuroPLC_Weights".w1[99] * v2[3] + "NeuroPLC_Weights".w1[100] * v2[4] + "NeuroPLC_Weights".w1[101] * v2[5] + "NeuroPLC_Weights".w1[102] * v2[6] + "NeuroPLC_Weights".w1[103] * v2[7] + "NeuroPLC_Weights".w1[104] * v2[8] + "NeuroPLC_Weights".w1[105] * v2[9] + "NeuroPLC_Weights".w1[106] * v2[10] + "NeuroPLC_Weights".w1[107] * v2[11] + "NeuroPLC_Weights".w1[108] * v2[12] + "NeuroPLC_Weights".w1[109] * v2[13] + "NeuroPLC_Weights".w1[110] * v2[14] + "NeuroPLC_Weights".w1[111] * v2[15] + "NeuroPLC_Weights".w1[112] * v2[16] + "NeuroPLC_Weights".w1[113] * v2[17] + "NeuroPLC_Weights".w1[114] * v2[18] + "NeuroPLC_Weights".w1[115] * v2[19] + "NeuroPLC_Weights".w1[116] * v2[20] + "NeuroPLC_Weights".w1[117] * v2[21] + "NeuroPLC_Weights".w1[118] * v2[22] + "NeuroPLC_Weights".w1[119] * v2[23] + "NeuroPLC_Weights".w1[120] * v2[24] + "NeuroPLC_Weights".w1[121] * v2[25] + "NeuroPLC_Weights".w1[122] * v2[26] + "NeuroPLC_Weights".w1[123] * v2[27] + "NeuroPLC_Weights".w1[124] * v2[28] + "NeuroPLC_Weights".w1[125] * v2[29] + "NeuroPLC_Weights".w1[126] * v2[30] + "NeuroPLC_Weights".w1[127] * v2[31];
    v3[4] := "NeuroPLC_Weights".w1[512 + 4] + "NeuroPLC_Weights".w1[128] * v2[0] + "NeuroPLC_Weights".w1[129] * v2[1] + "NeuroPLC_Weights".w1[130] * v2[2] + "NeuroPLC_Weights".w1[131] * v2[3] + "NeuroPLC_Weights".w1[132] * v2[4] + "NeuroPLC_Weights".w1[133] * v2[5] + "NeuroPLC_Weights".w1[134] * v2[6] + "NeuroPLC_Weights".w1[135] * v2[7] + "NeuroPLC_Weights".w1[136] * v2[8] + "NeuroPLC_Weights".w1[137] * v2[9] + "NeuroPLC_Weights".w1[138] * v2[10] + "NeuroPLC_Weights".w1[139] * v2[11] + "NeuroPLC_Weights".w1[140] * v2[12] + "NeuroPLC_Weights".w1[141] * v2[13] + "NeuroPLC_Weights".w1[142] * v2[14] + "NeuroPLC_Weights".w1[143] * v2[15] + "NeuroPLC_Weights".w1[144] * v2[16] + "NeuroPLC_Weights".w1[145] * v2[17] + "NeuroPLC_Weights".w1[146] * v2[18] + "NeuroPLC_Weights".w1[147] * v2[19] + "NeuroPLC_Weights".w1[148] * v2[20] + "NeuroPLC_Weights".w1[149] * v2[21] + "NeuroPLC_Weights".w1[150] * v2[22] + "NeuroPLC_Weights".w1[151] * v2[23] + "NeuroPLC_Weights".w1[152] * v2[24] + "NeuroPLC_Weights".w1[153] * v2[25] + "NeuroPLC_Weights".w1[154] * v2[26] + "NeuroPLC_Weights".w1[155] * v2[27] + "NeuroPLC_Weights".w1[156] * v2[28] + "NeuroPLC_Weights".w1[157] * v2[29] + "NeuroPLC_Weights".w1[158] * v2[30] + "NeuroPLC_Weights".w1[159] * v2[31];
    v3[5] := "NeuroPLC_Weights".w1[512 + 5] + "NeuroPLC_Weights".w1[160] * v2[0] + "NeuroPLC_Weights".w1[161] * v2[1] + "NeuroPLC_Weights".w1[162] * v2[2] + "NeuroPLC_Weights".w1[163] * v2[3] + "NeuroPLC_Weights".w1[164] * v2[4] + "NeuroPLC_Weights".w1[165] * v2[5] + "NeuroPLC_Weights".w1[166] * v2[6] + "NeuroPLC_Weights".w1[167] * v2[7] + "NeuroPLC_Weights".w1[168] * v2[8] + "NeuroPLC_Weights".w1[169] * v2[9] + "NeuroPLC_Weights".w1[170] * v2[10] + "NeuroPLC_Weights".w1[171] * v2[11] + "NeuroPLC_Weights".w1[172] * v2[12] + "NeuroPLC_Weights".w1[173] * v2[13] + "NeuroPLC_Weights".w1[174] * v2[14] + "NeuroPLC_Weights".w1[175] * v2[15] + "NeuroPLC_Weights".w1[176] * v2[16] + "NeuroPLC_Weights".w1[177] * v2[17] + "NeuroPLC_Weights".w1[178] * v2[18] + "NeuroPLC_Weights".w1[179] * v2[19] + "NeuroPLC_Weights".w1[180] * v2[20] + "NeuroPLC_Weights".w1[181] * v2[21] + "NeuroPLC_Weights".w1[182] * v2[22] + "NeuroPLC_Weights".w1[183] * v2[23] + "NeuroPLC_Weights".w1[184] * v2[24] + "NeuroPLC_Weights".w1[185] * v2[25] + "NeuroPLC_Weights".w1[186] * v2[26] + "NeuroPLC_Weights".w1[187] * v2[27] + "NeuroPLC_Weights".w1[188] * v2[28] + "NeuroPLC_Weights".w1[189] * v2[29] + "NeuroPLC_Weights".w1[190] * v2[30] + "NeuroPLC_Weights".w1[191] * v2[31];
    v3[6] := "NeuroPLC_Weights".w1[512 + 6] + "NeuroPLC_Weights".w1[192] * v2[0] + "NeuroPLC_Weights".w1[193] * v2[1] + "NeuroPLC_Weights".w1[194] * v2[2] + "NeuroPLC_Weights".w1[195] * v2[3] + "NeuroPLC_Weights".w1[196] * v2[4] + "NeuroPLC_Weights".w1[197] * v2[5] + "NeuroPLC_Weights".w1[198] * v2[6] + "NeuroPLC_Weights".w1[199] * v2[7] + "NeuroPLC_Weights".w1[200] * v2[8] + "NeuroPLC_Weights".w1[201] * v2[9] + "NeuroPLC_Weights".w1[202] * v2[10] + "NeuroPLC_Weights".w1[203] * v2[11] + "NeuroPLC_Weights".w1[204] * v2[12] + "NeuroPLC_Weights".w1[205] * v2[13] + "NeuroPLC_Weights".w1[206] * v2[14] + "NeuroPLC_Weights".w1[207] * v2[15] + "NeuroPLC_Weights".w1[208] * v2[16] + "NeuroPLC_Weights".w1[209] * v2[17] + "NeuroPLC_Weights".w1[210] * v2[18] + "NeuroPLC_Weights".w1[211] * v2[19] + "NeuroPLC_Weights".w1[212] * v2[20] + "NeuroPLC_Weights".w1[213] * v2[21] + "NeuroPLC_Weights".w1[214] * v2[22] + "NeuroPLC_Weights".w1[215] * v2[23] + "NeuroPLC_Weights".w1[216] * v2[24] + "NeuroPLC_Weights".w1[217] * v2[25] + "NeuroPLC_Weights".w1[218] * v2[26] + "NeuroPLC_Weights".w1[219] * v2[27] + "NeuroPLC_Weights".w1[220] * v2[28] + "NeuroPLC_Weights".w1[221] * v2[29] + "NeuroPLC_Weights".w1[222] * v2[30] + "NeuroPLC_Weights".w1[223] * v2[31];
    v3[7] := "NeuroPLC_Weights".w1[512 + 7] + "NeuroPLC_Weights".w1[224] * v2[0] + "NeuroPLC_Weights".w1[225] * v2[1] + "NeuroPLC_Weights".w1[226] * v2[2] + "NeuroPLC_Weights".w1[227] * v2[3] + "NeuroPLC_Weights".w1[228] * v2[4] + "NeuroPLC_Weights".w1[229] * v2[5] + "NeuroPLC_Weights".w1[230] * v2[6] + "NeuroPLC_Weights".w1[231] * v2[7] + "NeuroPLC_Weights".w1[232] * v2[8] + "NeuroPLC_Weights".w1[233] * v2[9] + "NeuroPLC_Weights".w1[234] * v2[10] + "NeuroPLC_Weights".w1[235] * v2[11] + "NeuroPLC_Weights".w1[236] * v2[12] + "NeuroPLC_Weights".w1[237] * v2[13] + "NeuroPLC_Weights".w1[238] * v2[14] + "NeuroPLC_Weights".w1[239] * v2[15] + "NeuroPLC_Weights".w1[240] * v2[16] + "NeuroPLC_Weights".w1[241] * v2[17] + "NeuroPLC_Weights".w1[242] * v2[18] + "NeuroPLC_Weights".w1[243] * v2[19] + "NeuroPLC_Weights".w1[244] * v2[20] + "NeuroPLC_Weights".w1[245] * v2[21] + "NeuroPLC_Weights".w1[246] * v2[22] + "NeuroPLC_Weights".w1[247] * v2[23] + "NeuroPLC_Weights".w1[248] * v2[24] + "NeuroPLC_Weights".w1[249] * v2[25] + "NeuroPLC_Weights".w1[250] * v2[26] + "NeuroPLC_Weights".w1[251] * v2[27] + "NeuroPLC_Weights".w1[252] * v2[28] + "NeuroPLC_Weights".w1[253] * v2[29] + "NeuroPLC_Weights".w1[254] * v2[30] + "NeuroPLC_Weights".w1[255] * v2[31];
    v3[8] := "NeuroPLC_Weights".w1[512 + 8] + "NeuroPLC_Weights".w1[256] * v2[0] + "NeuroPLC_Weights".w1[257] * v2[1] + "NeuroPLC_Weights".w1[258] * v2[2] + "NeuroPLC_Weights".w1[259] * v2[3] + "NeuroPLC_Weights".w1[260] * v2[4] + "NeuroPLC_Weights".w1[261] * v2[5] + "NeuroPLC_Weights".w1[262] * v2[6] + "NeuroPLC_Weights".w1[263] * v2[7] + "NeuroPLC_Weights".w1[264] * v2[8] + "NeuroPLC_Weights".w1[265] * v2[9] + "NeuroPLC_Weights".w1[266] * v2[10] + "NeuroPLC_Weights".w1[267] * v2[11] + "NeuroPLC_Weights".w1[268] * v2[12] + "NeuroPLC_Weights".w1[269] * v2[13] + "NeuroPLC_Weights".w1[270] * v2[14] + "NeuroPLC_Weights".w1[271] * v2[15] + "NeuroPLC_Weights".w1[272] * v2[16] + "NeuroPLC_Weights".w1[273] * v2[17] + "NeuroPLC_Weights".w1[274] * v2[18] + "NeuroPLC_Weights".w1[275] * v2[19] + "NeuroPLC_Weights".w1[276] * v2[20] + "NeuroPLC_Weights".w1[277] * v2[21] + "NeuroPLC_Weights".w1[278] * v2[22] + "NeuroPLC_Weights".w1[279] * v2[23] + "NeuroPLC_Weights".w1[280] * v2[24] + "NeuroPLC_Weights".w1[281] * v2[25] + "NeuroPLC_Weights".w1[282] * v2[26] + "NeuroPLC_Weights".w1[283] * v2[27] + "NeuroPLC_Weights".w1[284] * v2[28] + "NeuroPLC_Weights".w1[285] * v2[29] + "NeuroPLC_Weights".w1[286] * v2[30] + "NeuroPLC_Weights".w1[287] * v2[31];
    v3[9] := "NeuroPLC_Weights".w1[512 + 9] + "NeuroPLC_Weights".w1[288] * v2[0] + "NeuroPLC_Weights".w1[289] * v2[1] + "NeuroPLC_Weights".w1[290] * v2[2] + "NeuroPLC_Weights".w1[291] * v2[3] + "NeuroPLC_Weights".w1[292] * v2[4] + "NeuroPLC_Weights".w1[293] * v2[5] + "NeuroPLC_Weights".w1[294] * v2[6] + "NeuroPLC_Weights".w1[295] * v2[7] + "NeuroPLC_Weights".w1[296] * v2[8] + "NeuroPLC_Weights".w1[297] * v2[9] + "NeuroPLC_Weights".w1[298] * v2[10] + "NeuroPLC_Weights".w1[299] * v2[11] + "NeuroPLC_Weights".w1[300] * v2[12] + "NeuroPLC_Weights".w1[301] * v2[13] + "NeuroPLC_Weights".w1[302] * v2[14] + "NeuroPLC_Weights".w1[303] * v2[15] + "NeuroPLC_Weights".w1[304] * v2[16] + "NeuroPLC_Weights".w1[305] * v2[17] + "NeuroPLC_Weights".w1[306] * v2[18] + "NeuroPLC_Weights".w1[307] * v2[19] + "NeuroPLC_Weights".w1[308] * v2[20] + "NeuroPLC_Weights".w1[309] * v2[21] + "NeuroPLC_Weights".w1[310] * v2[22] + "NeuroPLC_Weights".w1[311] * v2[23] + "NeuroPLC_Weights".w1[312] * v2[24] + "NeuroPLC_Weights".w1[313] * v2[25] + "NeuroPLC_Weights".w1[314] * v2[26] + "NeuroPLC_Weights".w1[315] * v2[27] + "NeuroPLC_Weights".w1[316] * v2[28] + "NeuroPLC_Weights".w1[317] * v2[29] + "NeuroPLC_Weights".w1[318] * v2[30] + "NeuroPLC_Weights".w1[319] * v2[31];
    v3[10] := "NeuroPLC_Weights".w1[512 + 10] + "NeuroPLC_Weights".w1[320] * v2[0] + "NeuroPLC_Weights".w1[321] * v2[1] + "NeuroPLC_Weights".w1[322] * v2[2] + "NeuroPLC_Weights".w1[323] * v2[3] + "NeuroPLC_Weights".w1[324] * v2[4] + "NeuroPLC_Weights".w1[325] * v2[5] + "NeuroPLC_Weights".w1[326] * v2[6] + "NeuroPLC_Weights".w1[327] * v2[7] + "NeuroPLC_Weights".w1[328] * v2[8] + "NeuroPLC_Weights".w1[329] * v2[9] + "NeuroPLC_Weights".w1[330] * v2[10] + "NeuroPLC_Weights".w1[331] * v2[11] + "NeuroPLC_Weights".w1[332] * v2[12] + "NeuroPLC_Weights".w1[333] * v2[13] + "NeuroPLC_Weights".w1[334] * v2[14] + "NeuroPLC_Weights".w1[335] * v2[15] + "NeuroPLC_Weights".w1[336] * v2[16] + "NeuroPLC_Weights".w1[337] * v2[17] + "NeuroPLC_Weights".w1[338] * v2[18] + "NeuroPLC_Weights".w1[339] * v2[19] + "NeuroPLC_Weights".w1[340] * v2[20] + "NeuroPLC_Weights".w1[341] * v2[21] + "NeuroPLC_Weights".w1[342] * v2[22] + "NeuroPLC_Weights".w1[343] * v2[23] + "NeuroPLC_Weights".w1[344] * v2[24] + "NeuroPLC_Weights".w1[345] * v2[25] + "NeuroPLC_Weights".w1[346] * v2[26] + "NeuroPLC_Weights".w1[347] * v2[27] + "NeuroPLC_Weights".w1[348] * v2[28] + "NeuroPLC_Weights".w1[349] * v2[29] + "NeuroPLC_Weights".w1[350] * v2[30] + "NeuroPLC_Weights".w1[351] * v2[31];
    v3[11] := "NeuroPLC_Weights".w1[512 + 11] + "NeuroPLC_Weights".w1[352] * v2[0] + "NeuroPLC_Weights".w1[353] * v2[1] + "NeuroPLC_Weights".w1[354] * v2[2] + "NeuroPLC_Weights".w1[355] * v2[3] + "NeuroPLC_Weights".w1[356] * v2[4] + "NeuroPLC_Weights".w1[357] * v2[5] + "NeuroPLC_Weights".w1[358] * v2[6] + "NeuroPLC_Weights".w1[359] * v2[7] + "NeuroPLC_Weights".w1[360] * v2[8] + "NeuroPLC_Weights".w1[361] * v2[9] + "NeuroPLC_Weights".w1[362] * v2[10] + "NeuroPLC_Weights".w1[363] * v2[11] + "NeuroPLC_Weights".w1[364] * v2[12] + "NeuroPLC_Weights".w1[365] * v2[13] + "NeuroPLC_Weights".w1[366] * v2[14] + "NeuroPLC_Weights".w1[367] * v2[15] + "NeuroPLC_Weights".w1[368] * v2[16] + "NeuroPLC_Weights".w1[369] * v2[17] + "NeuroPLC_Weights".w1[370] * v2[18] + "NeuroPLC_Weights".w1[371] * v2[19] + "NeuroPLC_Weights".w1[372] * v2[20] + "NeuroPLC_Weights".w1[373] * v2[21] + "NeuroPLC_Weights".w1[374] * v2[22] + "NeuroPLC_Weights".w1[375] * v2[23] + "NeuroPLC_Weights".w1[376] * v2[24] + "NeuroPLC_Weights".w1[377] * v2[25] + "NeuroPLC_Weights".w1[378] * v2[26] + "NeuroPLC_Weights".w1[379] * v2[27] + "NeuroPLC_Weights".w1[380] * v2[28] + "NeuroPLC_Weights".w1[381] * v2[29] + "NeuroPLC_Weights".w1[382] * v2[30] + "NeuroPLC_Weights".w1[383] * v2[31];
    v3[12] := "NeuroPLC_Weights".w1[512 + 12] + "NeuroPLC_Weights".w1[384] * v2[0] + "NeuroPLC_Weights".w1[385] * v2[1] + "NeuroPLC_Weights".w1[386] * v2[2] + "NeuroPLC_Weights".w1[387] * v2[3] + "NeuroPLC_Weights".w1[388] * v2[4] + "NeuroPLC_Weights".w1[389] * v2[5] + "NeuroPLC_Weights".w1[390] * v2[6] + "NeuroPLC_Weights".w1[391] * v2[7] + "NeuroPLC_Weights".w1[392] * v2[8] + "NeuroPLC_Weights".w1[393] * v2[9] + "NeuroPLC_Weights".w1[394] * v2[10] + "NeuroPLC_Weights".w1[395] * v2[11] + "NeuroPLC_Weights".w1[396] * v2[12] + "NeuroPLC_Weights".w1[397] * v2[13] + "NeuroPLC_Weights".w1[398] * v2[14] + "NeuroPLC_Weights".w1[399] * v2[15] + "NeuroPLC_Weights".w1[400] * v2[16] + "NeuroPLC_Weights".w1[401] * v2[17] + "NeuroPLC_Weights".w1[402] * v2[18] + "NeuroPLC_Weights".w1[403] * v2[19] + "NeuroPLC_Weights".w1[404] * v2[20] + "NeuroPLC_Weights".w1[405] * v2[21] + "NeuroPLC_Weights".w1[406] * v2[22] + "NeuroPLC_Weights".w1[407] * v2[23] + "NeuroPLC_Weights".w1[408] * v2[24] + "NeuroPLC_Weights".w1[409] * v2[25] + "NeuroPLC_Weights".w1[410] * v2[26] + "NeuroPLC_Weights".w1[411] * v2[27] + "NeuroPLC_Weights".w1[412] * v2[28] + "NeuroPLC_Weights".w1[413] * v2[29] + "NeuroPLC_Weights".w1[414] * v2[30] + "NeuroPLC_Weights".w1[415] * v2[31];
    v3[13] := "NeuroPLC_Weights".w1[512 + 13] + "NeuroPLC_Weights".w1[416] * v2[0] + "NeuroPLC_Weights".w1[417] * v2[1] + "NeuroPLC_Weights".w1[418] * v2[2] + "NeuroPLC_Weights".w1[419] * v2[3] + "NeuroPLC_Weights".w1[420] * v2[4] + "NeuroPLC_Weights".w1[421] * v2[5] + "NeuroPLC_Weights".w1[422] * v2[6] + "NeuroPLC_Weights".w1[423] * v2[7] + "NeuroPLC_Weights".w1[424] * v2[8] + "NeuroPLC_Weights".w1[425] * v2[9] + "NeuroPLC_Weights".w1[426] * v2[10] + "NeuroPLC_Weights".w1[427] * v2[11] + "NeuroPLC_Weights".w1[428] * v2[12] + "NeuroPLC_Weights".w1[429] * v2[13] + "NeuroPLC_Weights".w1[430] * v2[14] + "NeuroPLC_Weights".w1[431] * v2[15] + "NeuroPLC_Weights".w1[432] * v2[16] + "NeuroPLC_Weights".w1[433] * v2[17] + "NeuroPLC_Weights".w1[434] * v2[18] + "NeuroPLC_Weights".w1[435] * v2[19] + "NeuroPLC_Weights".w1[436] * v2[20] + "NeuroPLC_Weights".w1[437] * v2[21] + "NeuroPLC_Weights".w1[438] * v2[22] + "NeuroPLC_Weights".w1[439] * v2[23] + "NeuroPLC_Weights".w1[440] * v2[24] + "NeuroPLC_Weights".w1[441] * v2[25] + "NeuroPLC_Weights".w1[442] * v2[26] + "NeuroPLC_Weights".w1[443] * v2[27] + "NeuroPLC_Weights".w1[444] * v2[28] + "NeuroPLC_Weights".w1[445] * v2[29] + "NeuroPLC_Weights".w1[446] * v2[30] + "NeuroPLC_Weights".w1[447] * v2[31];
    v3[14] := "NeuroPLC_Weights".w1[512 + 14] + "NeuroPLC_Weights".w1[448] * v2[0] + "NeuroPLC_Weights".w1[449] * v2[1] + "NeuroPLC_Weights".w1[450] * v2[2] + "NeuroPLC_Weights".w1[451] * v2[3] + "NeuroPLC_Weights".w1[452] * v2[4] + "NeuroPLC_Weights".w1[453] * v2[5] + "NeuroPLC_Weights".w1[454] * v2[6] + "NeuroPLC_Weights".w1[455] * v2[7] + "NeuroPLC_Weights".w1[456] * v2[8] + "NeuroPLC_Weights".w1[457] * v2[9] + "NeuroPLC_Weights".w1[458] * v2[10] + "NeuroPLC_Weights".w1[459] * v2[11] + "NeuroPLC_Weights".w1[460] * v2[12] + "NeuroPLC_Weights".w1[461] * v2[13] + "NeuroPLC_Weights".w1[462] * v2[14] + "NeuroPLC_Weights".w1[463] * v2[15] + "NeuroPLC_Weights".w1[464] * v2[16] + "NeuroPLC_Weights".w1[465] * v2[17] + "NeuroPLC_Weights".w1[466] * v2[18] + "NeuroPLC_Weights".w1[467] * v2[19] + "NeuroPLC_Weights".w1[468] * v2[20] + "NeuroPLC_Weights".w1[469] * v2[21] + "NeuroPLC_Weights".w1[470] * v2[22] + "NeuroPLC_Weights".w1[471] * v2[23] + "NeuroPLC_Weights".w1[472] * v2[24] + "NeuroPLC_Weights".w1[473] * v2[25] + "NeuroPLC_Weights".w1[474] * v2[26] + "NeuroPLC_Weights".w1[475] * v2[27] + "NeuroPLC_Weights".w1[476] * v2[28] + "NeuroPLC_Weights".w1[477] * v2[29] + "NeuroPLC_Weights".w1[478] * v2[30] + "NeuroPLC_Weights".w1[479] * v2[31];
    v3[15] := "NeuroPLC_Weights".w1[512 + 15] + "NeuroPLC_Weights".w1[480] * v2[0] + "NeuroPLC_Weights".w1[481] * v2[1] + "NeuroPLC_Weights".w1[482] * v2[2] + "NeuroPLC_Weights".w1[483] * v2[3] + "NeuroPLC_Weights".w1[484] * v2[4] + "NeuroPLC_Weights".w1[485] * v2[5] + "NeuroPLC_Weights".w1[486] * v2[6] + "NeuroPLC_Weights".w1[487] * v2[7] + "NeuroPLC_Weights".w1[488] * v2[8] + "NeuroPLC_Weights".w1[489] * v2[9] + "NeuroPLC_Weights".w1[490] * v2[10] + "NeuroPLC_Weights".w1[491] * v2[11] + "NeuroPLC_Weights".w1[492] * v2[12] + "NeuroPLC_Weights".w1[493] * v2[13] + "NeuroPLC_Weights".w1[494] * v2[14] + "NeuroPLC_Weights".w1[495] * v2[15] + "NeuroPLC_Weights".w1[496] * v2[16] + "NeuroPLC_Weights".w1[497] * v2[17] + "NeuroPLC_Weights".w1[498] * v2[18] + "NeuroPLC_Weights".w1[499] * v2[19] + "NeuroPLC_Weights".w1[500] * v2[20] + "NeuroPLC_Weights".w1[501] * v2[21] + "NeuroPLC_Weights".w1[502] * v2[22] + "NeuroPLC_Weights".w1[503] * v2[23] + "NeuroPLC_Weights".w1[504] * v2[24] + "NeuroPLC_Weights".w1[505] * v2[25] + "NeuroPLC_Weights".w1[506] * v2[26] + "NeuroPLC_Weights".w1[507] * v2[27] + "NeuroPLC_Weights".w1[508] * v2[28] + "NeuroPLC_Weights".w1[509] * v2[29] + "NeuroPLC_Weights".w1[510] * v2[30] + "NeuroPLC_Weights".w1[511] * v2[31];

    // ---- relu1: RELU ----
    IF v3[0] > 0.0 THEN v4[0] := v3[0]; ELSE v4[0] := 0.0; END_IF;
    IF v3[1] > 0.0 THEN v4[1] := v3[1]; ELSE v4[1] := 0.0; END_IF;
    IF v3[2] > 0.0 THEN v4[2] := v3[2]; ELSE v4[2] := 0.0; END_IF;
    IF v3[3] > 0.0 THEN v4[3] := v3[3]; ELSE v4[3] := 0.0; END_IF;
    IF v3[4] > 0.0 THEN v4[4] := v3[4]; ELSE v4[4] := 0.0; END_IF;
    IF v3[5] > 0.0 THEN v4[5] := v3[5]; ELSE v4[5] := 0.0; END_IF;
    IF v3[6] > 0.0 THEN v4[6] := v3[6]; ELSE v4[6] := 0.0; END_IF;
    IF v3[7] > 0.0 THEN v4[7] := v3[7]; ELSE v4[7] := 0.0; END_IF;
    IF v3[8] > 0.0 THEN v4[8] := v3[8]; ELSE v4[8] := 0.0; END_IF;
    IF v3[9] > 0.0 THEN v4[9] := v3[9]; ELSE v4[9] := 0.0; END_IF;
    IF v3[10] > 0.0 THEN v4[10] := v3[10]; ELSE v4[10] := 0.0; END_IF;
    IF v3[11] > 0.0 THEN v4[11] := v3[11]; ELSE v4[11] := 0.0; END_IF;
    IF v3[12] > 0.0 THEN v4[12] := v3[12]; ELSE v4[12] := 0.0; END_IF;
    IF v3[13] > 0.0 THEN v4[13] := v3[13]; ELSE v4[13] := 0.0; END_IF;
    IF v3[14] > 0.0 THEN v4[14] := v3[14]; ELSE v4[14] := 0.0; END_IF;
    IF v3[15] > 0.0 THEN v4[15] := v3[15]; ELSE v4[15] := 0.0; END_IF;

    // ---- fc2: MatMul(16→4) ----
    // W = "NeuroPLC_Weights".w2[:64],   b = w2[64:]
    v5[0] := "NeuroPLC_Weights".w2[64 + 0] + "NeuroPLC_Weights".w2[0] * v4[0] + "NeuroPLC_Weights".w2[1] * v4[1] + "NeuroPLC_Weights".w2[2] * v4[2] + "NeuroPLC_Weights".w2[3] * v4[3] + "NeuroPLC_Weights".w2[4] * v4[4] + "NeuroPLC_Weights".w2[5] * v4[5] + "NeuroPLC_Weights".w2[6] * v4[6] + "NeuroPLC_Weights".w2[7] * v4[7] + "NeuroPLC_Weights".w2[8] * v4[8] + "NeuroPLC_Weights".w2[9] * v4[9] + "NeuroPLC_Weights".w2[10] * v4[10] + "NeuroPLC_Weights".w2[11] * v4[11] + "NeuroPLC_Weights".w2[12] * v4[12] + "NeuroPLC_Weights".w2[13] * v4[13] + "NeuroPLC_Weights".w2[14] * v4[14] + "NeuroPLC_Weights".w2[15] * v4[15];
    v5[1] := "NeuroPLC_Weights".w2[64 + 1] + "NeuroPLC_Weights".w2[16] * v4[0] + "NeuroPLC_Weights".w2[17] * v4[1] + "NeuroPLC_Weights".w2[18] * v4[2] + "NeuroPLC_Weights".w2[19] * v4[3] + "NeuroPLC_Weights".w2[20] * v4[4] + "NeuroPLC_Weights".w2[21] * v4[5] + "NeuroPLC_Weights".w2[22] * v4[6] + "NeuroPLC_Weights".w2[23] * v4[7] + "NeuroPLC_Weights".w2[24] * v4[8] + "NeuroPLC_Weights".w2[25] * v4[9] + "NeuroPLC_Weights".w2[26] * v4[10] + "NeuroPLC_Weights".w2[27] * v4[11] + "NeuroPLC_Weights".w2[28] * v4[12] + "NeuroPLC_Weights".w2[29] * v4[13] + "NeuroPLC_Weights".w2[30] * v4[14] + "NeuroPLC_Weights".w2[31] * v4[15];
    v5[2] := "NeuroPLC_Weights".w2[64 + 2] + "NeuroPLC_Weights".w2[32] * v4[0] + "NeuroPLC_Weights".w2[33] * v4[1] + "NeuroPLC_Weights".w2[34] * v4[2] + "NeuroPLC_Weights".w2[35] * v4[3] + "NeuroPLC_Weights".w2[36] * v4[4] + "NeuroPLC_Weights".w2[37] * v4[5] + "NeuroPLC_Weights".w2[38] * v4[6] + "NeuroPLC_Weights".w2[39] * v4[7] + "NeuroPLC_Weights".w2[40] * v4[8] + "NeuroPLC_Weights".w2[41] * v4[9] + "NeuroPLC_Weights".w2[42] * v4[10] + "NeuroPLC_Weights".w2[43] * v4[11] + "NeuroPLC_Weights".w2[44] * v4[12] + "NeuroPLC_Weights".w2[45] * v4[13] + "NeuroPLC_Weights".w2[46] * v4[14] + "NeuroPLC_Weights".w2[47] * v4[15];
    v5[3] := "NeuroPLC_Weights".w2[64 + 3] + "NeuroPLC_Weights".w2[48] * v4[0] + "NeuroPLC_Weights".w2[49] * v4[1] + "NeuroPLC_Weights".w2[50] * v4[2] + "NeuroPLC_Weights".w2[51] * v4[3] + "NeuroPLC_Weights".w2[52] * v4[4] + "NeuroPLC_Weights".w2[53] * v4[5] + "NeuroPLC_Weights".w2[54] * v4[6] + "NeuroPLC_Weights".w2[55] * v4[7] + "NeuroPLC_Weights".w2[56] * v4[8] + "NeuroPLC_Weights".w2[57] * v4[9] + "NeuroPLC_Weights".w2[58] * v4[10] + "NeuroPLC_Weights".w2[59] * v4[11] + "NeuroPLC_Weights".w2[60] * v4[12] + "NeuroPLC_Weights".w2[61] * v4[13] + "NeuroPLC_Weights".w2[62] * v4[14] + "NeuroPLC_Weights".w2[63] * v4[15];

    // ---- softmax: Softmax ----
    softmax_out[0] := EXP(v5[0]);
    softmax_out[1] := EXP(v5[1]);
    softmax_out[2] := EXP(v5[2]);
    softmax_out[3] := EXP(v5[3]);
    sum_val := softmax_out[0]
             + softmax_out[1]
             + softmax_out[2]
             + softmax_out[3]
             ;
    IF sum_val > 0.0 THEN
        softmax_out[0] := softmax_out[0] / sum_val;
        softmax_out[1] := softmax_out[1] / sum_val;
        softmax_out[2] := softmax_out[2] / sum_val;
        softmax_out[3] := softmax_out[3] / sum_val;
    END_IF;

    // ---- Argmax ----
    max_val := softmax_out[0];
    fault_class := 0;
    IF softmax_out[1] > max_val THEN
        max_val := softmax_out[1];
        fault_class := 1;
    END_IF;
    IF softmax_out[2] > max_val THEN
        max_val := softmax_out[2];
        fault_class := 2;
    END_IF;
    IF softmax_out[3] > max_val THEN
        max_val := softmax_out[3];
        fault_class := 3;
    END_IF;
    confidence := max_val;

END_FUNCTION_BLOCK